REGION Network 66: UNIT 2 STATION 3 COAXIAL CAMERA START NOZZLE ANALISIS METHOD WORKING OR BLOCKED ALARM
   RUNG wire#powerrail
      Contact( "DB16345_U2_STA3_CAM_NOZZLE_ANALISIS_TRIG".Done )
      { S7_Templates := "SrcType := Int" } NE_Contact(in1 := "DB16005_U2_STA3_COAXIAL_CLIENT_INTERFACE".U2_STA3_CAM_Analysis."Analyze nozzle".Outputs.Result, in2 := 0)
      wire#w1
      Contact( "DB7257_UNIT_2_STA_3_COAXIAL_ENABLE_DISABLE".ENABLED )
      wire#w2
      Coil( "DB16000_OPC_UA_TRIGGER_ALARM".CLIENT.U2_STA3_COAXIAL.ALARMS.CAM_START_NOZZLE_ANALISIS_METHOD_WORKING_BLOCKED_A )
   END_RUNG
   RUNG wire#powerrail
      Contact( "DB16000_OPC_UA_TRIGGER_ALARM".CLIENT.U2_STA3_COAXIAL.ALARMS.CAM_START_NOZZLE_ANALISIS_METHOD_WORKING_BLOCKED_A )
      I_Contact( "DB2120_MPP_ITC_IPC".RESET_FAULTS )
   END_RUNG wire#w1
   RUNG wire#w2
      Coil( "DB426_ALARMS_WARNINGS".ALARMS.UNIT_02.STATION_3_COAXIAL."720913" )
   END_RUNG
   // the same network as SCL:
   "DB16000_OPC_UA_TRIGGER_ALARM".CLIENT.U2_STA3_COAXIAL.ALARMS.CAM_START_NOZZLE_ANALISIS_METHOD_WORKING_BLOCKED_A := (("DB16345_U2_STA3_CAM_NOZZLE_ANALISIS_TRIG".Done AND ("DB16005_U2_STA3_COAXIAL_CLIENT_INTERFACE".U2_STA3_CAM_Analysis."Analyze nozzle".Outputs.Result <> 0)) OR ("DB16000_OPC_UA_TRIGGER_ALARM".CLIENT.U2_STA3_COAXIAL.ALARMS.CAM_START_NOZZLE_ANALISIS_METHOD_WORKING_BLOCKED_A AND NOT "DB2120_MPP_ITC_IPC".RESET_FAULTS)) AND "DB7257_UNIT_2_STA_3_COAXIAL_ENABLE_DISABLE".ENABLED;
   "DB426_ALARMS_WARNINGS".ALARMS.UNIT_02.STATION_3_COAXIAL."720913" := "DB16000_OPC_UA_TRIGGER_ALARM".CLIENT.U2_STA3_COAXIAL.ALARMS.CAM_START_NOZZLE_ANALISIS_METHOD_WORKING_BLOCKED_A;
END_REGION

REGION Network 67: UNIT 2 STATION 3 COAXIAL CAMERA START JET ANALISIS METHOD CONNECTION ALARM
   RUNG wire#powerrail
      Contact( "DB16346_U2_STA3_CAM_JET_ANALISIS_TRIG".Error )
      wire#w1
      Contact( "DB7257_UNIT_2_STA_3_COAXIAL_ENABLE_DISABLE".ENABLED )
      wire#w2
      Coil( "DB16000_OPC_UA_TRIGGER_ALARM".CLIENT.U2_STA3_COAXIAL.ALARMS.CAM_START_JET_ANALISIS_CONNECTION_A )
   END_RUNG
   RUNG wire#powerrail
      Contact( "DB16000_OPC_UA_TRIGGER_ALARM".CLIENT.U2_STA3_COAXIAL.ALARMS.CAM_START_JET_ANALISIS_CONNECTION_A )
      I_Contact( "DB2120_MPP_ITC_IPC".RESET_FAULTS )
   END_RUNG wire#w1
   RUNG wire#w2
      Coil( "DB426_ALARMS_WARNINGS".ALARMS.UNIT_02.STATION_3_COAXIAL."720920" )
   END_RUNG
   // the same network as SCL:
   "DB16000_OPC_UA_TRIGGER_ALARM".CLIENT.U2_STA3_COAXIAL.ALARMS.CAM_START_JET_ANALISIS_CONNECTION_A := ("DB16346_U2_STA3_CAM_JET_ANALISIS_TRIG".Error OR ("DB16000_OPC_UA_TRIGGER_ALARM".CLIENT.U2_STA3_COAXIAL.ALARMS.CAM_START_JET_ANALISIS_CONNECTION_A AND NOT "DB2120_MPP_ITC_IPC".RESET_FAULTS)) AND "DB7257_UNIT_2_STA_3_COAXIAL_ENABLE_DISABLE".ENABLED;
   "DB426_ALARMS_WARNINGS".ALARMS.UNIT_02.STATION_3_COAXIAL."720920" := "DB16000_OPC_UA_TRIGGER_ALARM".CLIENT.U2_STA3_COAXIAL.ALARMS.CAM_START_JET_ANALISIS_CONNECTION_A;
END_REGION

REGION Network 68: UNIT 2 STATION 3 COAXIAL CAMERA START JET ANALISIS METHOD WORKING OR BLOCKED ALARM
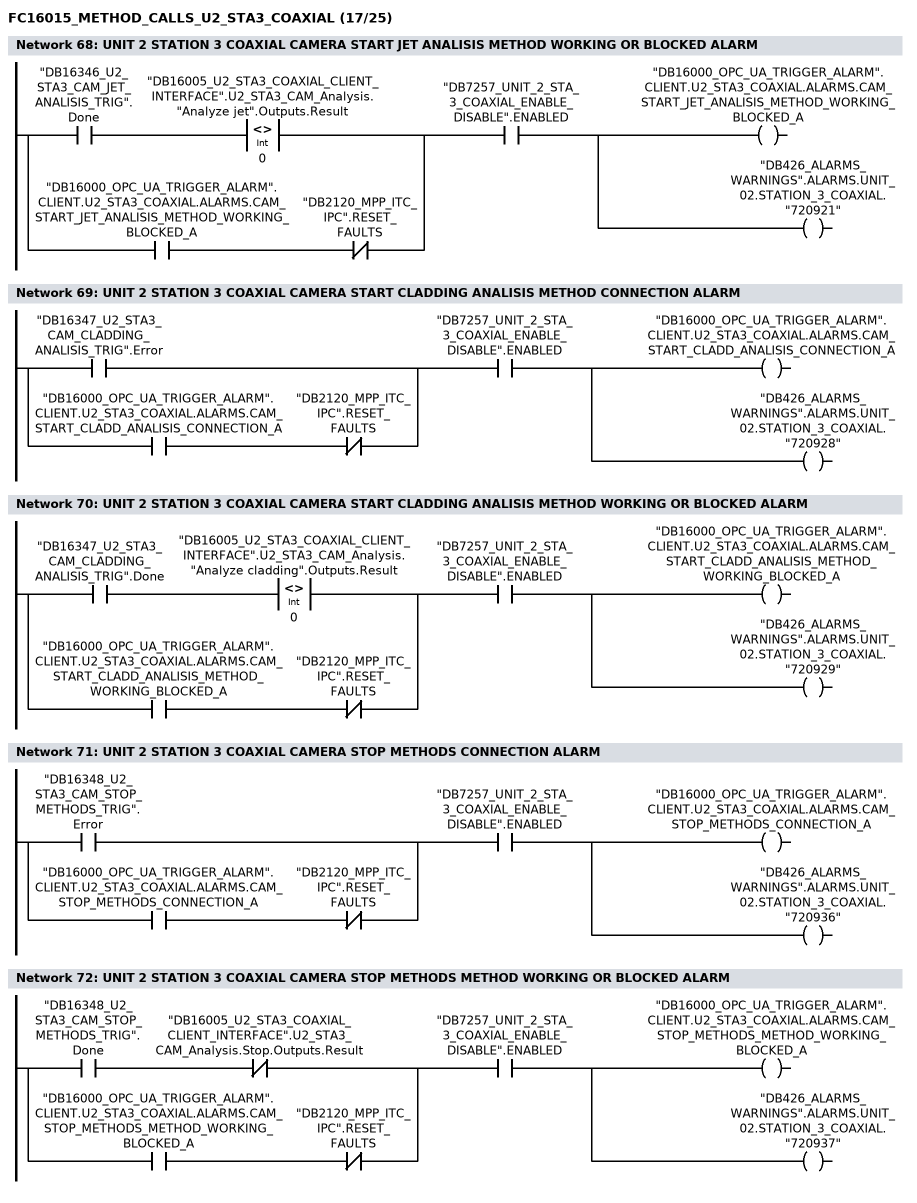
   RUNG wire#powerrail
      Contact( "DB16346_U2_STA3_CAM_JET_ANALISIS_TRIG".Done )
      { S7_Templates := "SrcType := Int" } NE_Contact(in1 := "DB16005_U2_STA3_COAXIAL_CLIENT_INTERFACE".U2_STA3_CAM_Analysis."Analyze jet".Outputs.Result, in2 := 0)
      wire#w1
      Contact( "DB7257_UNIT_2_STA_3_COAXIAL_ENABLE_DISABLE".ENABLED )
      wire#w2
      Coil( "DB16000_OPC_UA_TRIGGER_ALARM".CLIENT.U2_STA3_COAXIAL.ALARMS.CAM_START_JET_ANALISIS_METHOD_WORKING_BLOCKED_A )
   END_RUNG
   RUNG wire#powerrail
      Contact( "DB16000_OPC_UA_TRIGGER_ALARM".CLIENT.U2_STA3_COAXIAL.ALARMS.CAM_START_JET_ANALISIS_METHOD_WORKING_BLOCKED_A )
      I_Contact( "DB2120_MPP_ITC_IPC".RESET_FAULTS )
   END_RUNG wire#w1
   RUNG wire#w2
      Coil( "DB426_ALARMS_WARNINGS".ALARMS.UNIT_02.STATION_3_COAXIAL."720921" )
   END_RUNG
   // the same network as SCL:
   "DB16000_OPC_UA_TRIGGER_ALARM".CLIENT.U2_STA3_COAXIAL.ALARMS.CAM_START_JET_ANALISIS_METHOD_WORKING_BLOCKED_A := (("DB16346_U2_STA3_CAM_JET_ANALISIS_TRIG".Done AND ("DB16005_U2_STA3_COAXIAL_CLIENT_INTERFACE".U2_STA3_CAM_Analysis."Analyze jet".Outputs.Result <> 0)) OR ("DB16000_OPC_UA_TRIGGER_ALARM".CLIENT.U2_STA3_COAXIAL.ALARMS.CAM_START_JET_ANALISIS_METHOD_WORKING_BLOCKED_A AND NOT "DB2120_MPP_ITC_IPC".RESET_FAULTS)) AND "DB7257_UNIT_2_STA_3_COAXIAL_ENABLE_DISABLE".ENABLED;
   "DB426_ALARMS_WARNINGS".ALARMS.UNIT_02.STATION_3_COAXIAL."720921" := "DB16000_OPC_UA_TRIGGER_ALARM".CLIENT.U2_STA3_COAXIAL.ALARMS.CAM_START_JET_ANALISIS_METHOD_WORKING_BLOCKED_A;
END_REGION

REGION Network 69: UNIT 2 STATION 3 COAXIAL CAMERA START CLADDING ANALISIS METHOD CONNECTION ALARM
   RUNG wire#powerrail
      Contact( "DB16347_U2_STA3_CAM_CLADDING_ANALISIS_TRIG".Error )
      wire#w1
      Contact( "DB7257_UNIT_2_STA_3_COAXIAL_ENABLE_DISABLE".ENABLED )
      wire#w2
      Coil( "DB16000_OPC_UA_TRIGGER_ALARM".CLIENT.U2_STA3_COAXIAL.ALARMS.CAM_START_CLADD_ANALISIS_CONNECTION_A )
   END_RUNG
   RUNG wire#powerrail
      Contact( "DB16000_OPC_UA_TRIGGER_ALARM".CLIENT.U2_STA3_COAXIAL.ALARMS.CAM_START_CLADD_ANALISIS_CONNECTION_A )
      I_Contact( "DB2120_MPP_ITC_IPC".RESET_FAULTS )
   END_RUNG wire#w1
   RUNG wire#w2
      Coil( "DB426_ALARMS_WARNINGS".ALARMS.UNIT_02.STATION_3_COAXIAL."720928" )
   END_RUNG
   // the same network as SCL:
   "DB16000_OPC_UA_TRIGGER_ALARM".CLIENT.U2_STA3_COAXIAL.ALARMS.CAM_START_CLADD_ANALISIS_CONNECTION_A := ("DB16347_U2_STA3_CAM_CLADDING_ANALISIS_TRIG".Error OR ("DB16000_OPC_UA_TRIGGER_ALARM".CLIENT.U2_STA3_COAXIAL.ALARMS.CAM_START_CLADD_ANALISIS_CONNECTION_A AND NOT "DB2120_MPP_ITC_IPC".RESET_FAULTS)) AND "DB7257_UNIT_2_STA_3_COAXIAL_ENABLE_DISABLE".ENABLED;
   "DB426_ALARMS_WARNINGS".ALARMS.UNIT_02.STATION_3_COAXIAL."720928" := "DB16000_OPC_UA_TRIGGER_ALARM".CLIENT.U2_STA3_COAXIAL.ALARMS.CAM_START_CLADD_ANALISIS_CONNECTION_A;
END_REGION

REGION Network 70: UNIT 2 STATION 3 COAXIAL CAMERA START CLADDING ANALISIS METHOD WORKING OR BLOCKED ALARM
   RUNG wire#powerrail
      Contact( "DB16347_U2_STA3_CAM_CLADDING_ANALISIS_TRIG".Done )
      { S7_Templates := "SrcType := Int" } NE_Contact(in1 := "DB16005_U2_STA3_COAXIAL_CLIENT_INTERFACE".U2_STA3_CAM_Analysis."Analyze cladding".Outputs.Result, in2 := 0)
      wire#w1
      Contact( "DB7257_UNIT_2_STA_3_COAXIAL_ENABLE_DISABLE".ENABLED )
      wire#w2
      Coil( "DB16000_OPC_UA_TRIGGER_ALARM".CLIENT.U2_STA3_COAXIAL.ALARMS.CAM_START_CLADD_ANALISIS_METHOD_WORKING_BLOCKED_A )
   END_RUNG
   RUNG wire#powerrail
      Contact( "DB16000_OPC_UA_TRIGGER_ALARM".CLIENT.U2_STA3_COAXIAL.ALARMS.CAM_START_CLADD_ANALISIS_METHOD_WORKING_BLOCKED_A )
      I_Contact( "DB2120_MPP_ITC_IPC".RESET_FAULTS )
   END_RUNG wire#w1
   RUNG wire#w2
      Coil( "DB426_ALARMS_WARNINGS".ALARMS.UNIT_02.STATION_3_COAXIAL."720929" )
   END_RUNG
   // the same network as SCL:
   "DB16000_OPC_UA_TRIGGER_ALARM".CLIENT.U2_STA3_COAXIAL.ALARMS.CAM_START_CLADD_ANALISIS_METHOD_WORKING_BLOCKED_A := (("DB16347_U2_STA3_CAM_CLADDING_ANALISIS_TRIG".Done AND ("DB16005_U2_STA3_COAXIAL_CLIENT_INTERFACE".U2_STA3_CAM_Analysis."Analyze cladding".Outputs.Result <> 0)) OR ("DB16000_OPC_UA_TRIGGER_ALARM".CLIENT.U2_STA3_COAXIAL.ALARMS.CAM_START_CLADD_ANALISIS_METHOD_WORKING_BLOCKED_A AND NOT "DB2120_MPP_ITC_IPC".RESET_FAULTS)) AND "DB7257_UNIT_2_STA_3_COAXIAL_ENABLE_DISABLE".ENABLED;
   "DB426_ALARMS_WARNINGS".ALARMS.UNIT_02.STATION_3_COAXIAL."720929" := "DB16000_OPC_UA_TRIGGER_ALARM".CLIENT.U2_STA3_COAXIAL.ALARMS.CAM_START_CLADD_ANALISIS_METHOD_WORKING_BLOCKED_A;
END_REGION

REGION Network 71: UNIT 2 STATION 3 COAXIAL CAMERA STOP METHODS CONNECTION ALARM
   RUNG wire#powerrail
      Contact( "DB16348_U2_STA3_CAM_STOP_METHODS_TRIG".Error )
      wire#w1
      Contact( "DB7257_UNIT_2_STA_3_COAXIAL_ENABLE_DISABLE".ENABLED )
      wire#w2
      Coil( "DB16000_OPC_UA_TRIGGER_ALARM".CLIENT.U2_STA3_COAXIAL.ALARMS.CAM_STOP_METHODS_CONNECTION_A )
   END_RUNG
   RUNG wire#powerrail
      Contact( "DB16000_OPC_UA_TRIGGER_ALARM".CLIENT.U2_STA3_COAXIAL.ALARMS.CAM_STOP_METHODS_CONNECTION_A )
      I_Contact( "DB2120_MPP_ITC_IPC".RESET_FAULTS )
   END_RUNG wire#w1
   RUNG wire#w2
      Coil( "DB426_ALARMS_WARNINGS".ALARMS.UNIT_02.STATION_3_COAXIAL."720936" )
   END_RUNG
   // the same network as SCL:
   "DB16000_OPC_UA_TRIGGER_ALARM".CLIENT.U2_STA3_COAXIAL.ALARMS.CAM_STOP_METHODS_CONNECTION_A := ("DB16348_U2_STA3_CAM_STOP_METHODS_TRIG".Error OR ("DB16000_OPC_UA_TRIGGER_ALARM".CLIENT.U2_STA3_COAXIAL.ALARMS.CAM_STOP_METHODS_CONNECTION_A AND NOT "DB2120_MPP_ITC_IPC".RESET_FAULTS)) AND "DB7257_UNIT_2_STA_3_COAXIAL_ENABLE_DISABLE".ENABLED;
   "DB426_ALARMS_WARNINGS".ALARMS.UNIT_02.STATION_3_COAXIAL."720936" := "DB16000_OPC_UA_TRIGGER_ALARM".CLIENT.U2_STA3_COAXIAL.ALARMS.CAM_STOP_METHODS_CONNECTION_A;
END_REGION

REGION Network 72: UNIT 2 STATION 3 COAXIAL CAMERA STOP METHODS METHOD WORKING OR BLOCKED ALARM
   RUNG wire#powerrail
      Contact( "DB16348_U2_STA3_CAM_STOP_METHODS_TRIG".Done )
      I_Contact( "DB16005_U2_STA3_COAXIAL_CLIENT_INTERFACE".U2_STA3_CAM_Analysis.Stop.Outputs.Result )
      wire#w1
      Contact( "DB7257_UNIT_2_STA_3_COAXIAL_ENABLE_DISABLE".ENABLED )
      wire#w2
      Coil( "DB16000_OPC_UA_TRIGGER_ALARM".CLIENT.U2_STA3_COAXIAL.ALARMS.CAM_STOP_METHODS_METHOD_WORKING_BLOCKED_A )
   END_RUNG
   RUNG wire#powerrail
      Contact( "DB16000_OPC_UA_TRIGGER_ALARM".CLIENT.U2_STA3_COAXIAL.ALARMS.CAM_STOP_METHODS_METHOD_WORKING_BLOCKED_A )
      I_Contact( "DB2120_MPP_ITC_IPC".RESET_FAULTS )
   END_RUNG wire#w1
   RUNG wire#w2
      Coil( "DB426_ALARMS_WARNINGS".ALARMS.UNIT_02.STATION_3_COAXIAL."720937" )
   END_RUNG
   // the same network as SCL:
   "DB16000_OPC_UA_TRIGGER_ALARM".CLIENT.U2_STA3_COAXIAL.ALARMS.CAM_STOP_METHODS_METHOD_WORKING_BLOCKED_A := (("DB16348_U2_STA3_CAM_STOP_METHODS_TRIG".Done AND NOT "DB16005_U2_STA3_COAXIAL_CLIENT_INTERFACE".U2_STA3_CAM_Analysis.Stop.Outputs.Result) OR ("DB16000_OPC_UA_TRIGGER_ALARM".CLIENT.U2_STA3_COAXIAL.ALARMS.CAM_STOP_METHODS_METHOD_WORKING_BLOCKED_A AND NOT "DB2120_MPP_ITC_IPC".RESET_FAULTS)) AND "DB7257_UNIT_2_STA_3_COAXIAL_ENABLE_DISABLE".ENABLED;
   "DB426_ALARMS_WARNINGS".ALARMS.UNIT_02.STATION_3_COAXIAL."720937" := "DB16000_OPC_UA_TRIGGER_ALARM".CLIENT.U2_STA3_COAXIAL.ALARMS.CAM_STOP_METHODS_METHOD_WORKING_BLOCKED_A;
END_REGION

REGION Network 73: UNIT 2 STATION 3 COAXIAL CAMERA RESET PC METHOD CONNECTION ALARM
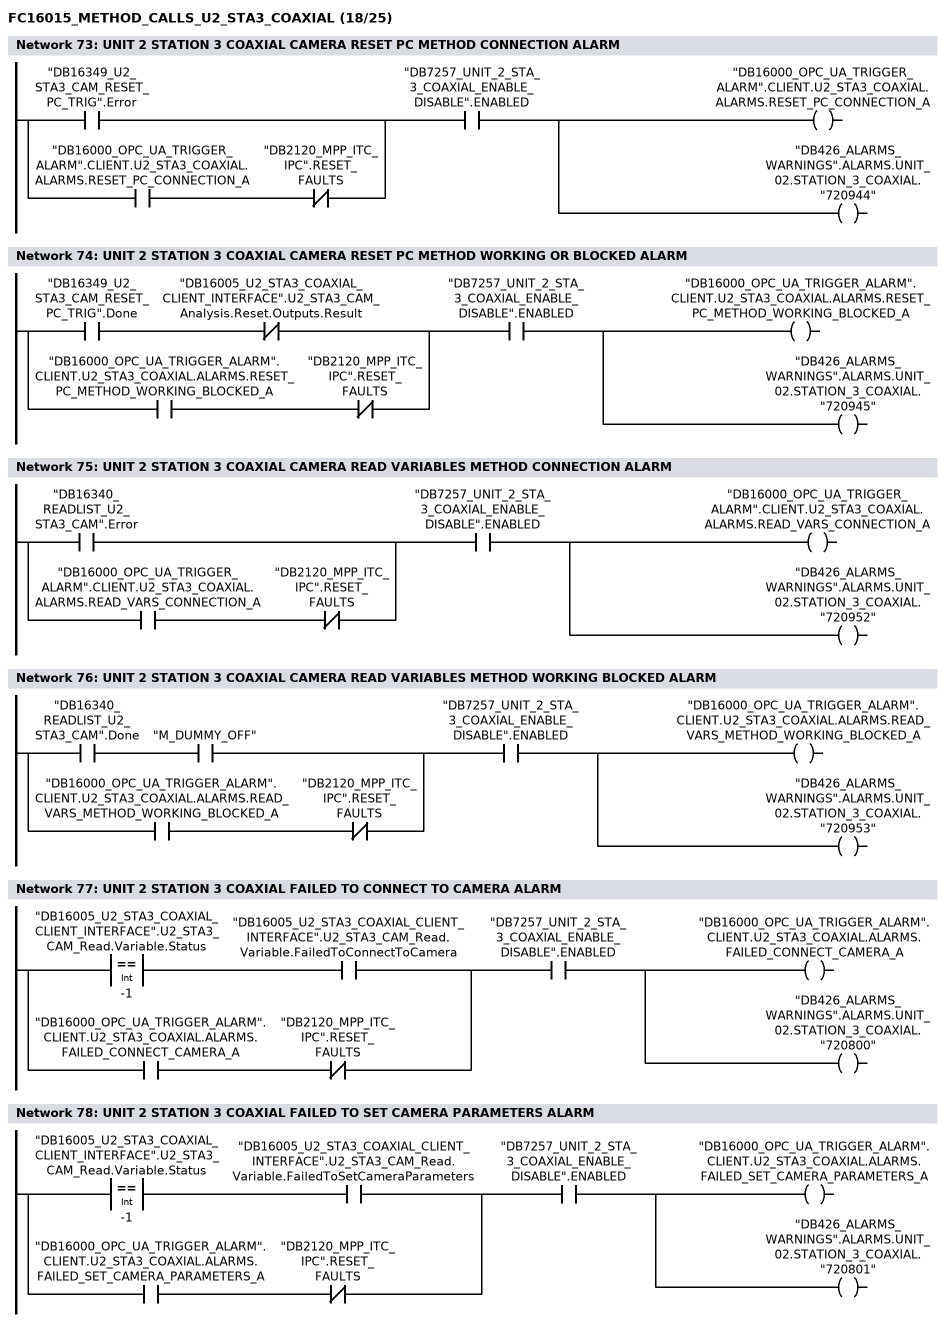
   RUNG wire#powerrail
      Contact( "DB16349_U2_STA3_CAM_RESET_PC_TRIG".Error )
      wire#w1
      Contact( "DB7257_UNIT_2_STA_3_COAXIAL_ENABLE_DISABLE".ENABLED )
      wire#w2
      Coil( "DB16000_OPC_UA_TRIGGER_ALARM".CLIENT.U2_STA3_COAXIAL.ALARMS.RESET_PC_CONNECTION_A )
   END_RUNG
   RUNG wire#powerrail
      Contact( "DB16000_OPC_UA_TRIGGER_ALARM".CLIENT.U2_STA3_COAXIAL.ALARMS.RESET_PC_CONNECTION_A )
      I_Contact( "DB2120_MPP_ITC_IPC".RESET_FAULTS )
   END_RUNG wire#w1
   RUNG wire#w2
      Coil( "DB426_ALARMS_WARNINGS".ALARMS.UNIT_02.STATION_3_COAXIAL."720944" )
   END_RUNG
   // the same network as SCL:
   "DB16000_OPC_UA_TRIGGER_ALARM".CLIENT.U2_STA3_COAXIAL.ALARMS.RESET_PC_CONNECTION_A := ("DB16349_U2_STA3_CAM_RESET_PC_TRIG".Error OR ("DB16000_OPC_UA_TRIGGER_ALARM".CLIENT.U2_STA3_COAXIAL.ALARMS.RESET_PC_CONNECTION_A AND NOT "DB2120_MPP_ITC_IPC".RESET_FAULTS)) AND "DB7257_UNIT_2_STA_3_COAXIAL_ENABLE_DISABLE".ENABLED;
   "DB426_ALARMS_WARNINGS".ALARMS.UNIT_02.STATION_3_COAXIAL."720944" := "DB16000_OPC_UA_TRIGGER_ALARM".CLIENT.U2_STA3_COAXIAL.ALARMS.RESET_PC_CONNECTION_A;
END_REGION

REGION Network 74: UNIT 2 STATION 3 COAXIAL CAMERA RESET PC METHOD WORKING OR BLOCKED ALARM
   RUNG wire#powerrail
      Contact( "DB16349_U2_STA3_CAM_RESET_PC_TRIG".Done )
      I_Contact( "DB16005_U2_STA3_COAXIAL_CLIENT_INTERFACE".U2_STA3_CAM_Analysis.Reset.Outputs.Result )
      wire#w1
      Contact( "DB7257_UNIT_2_STA_3_COAXIAL_ENABLE_DISABLE".ENABLED )
      wire#w2
      Coil( "DB16000_OPC_UA_TRIGGER_ALARM".CLIENT.U2_STA3_COAXIAL.ALARMS.RESET_PC_METHOD_WORKING_BLOCKED_A )
   END_RUNG
   RUNG wire#powerrail
      Contact( "DB16000_OPC_UA_TRIGGER_ALARM".CLIENT.U2_STA3_COAXIAL.ALARMS.RESET_PC_METHOD_WORKING_BLOCKED_A )
      I_Contact( "DB2120_MPP_ITC_IPC".RESET_FAULTS )
   END_RUNG wire#w1
   RUNG wire#w2
      Coil( "DB426_ALARMS_WARNINGS".ALARMS.UNIT_02.STATION_3_COAXIAL."720945" )
   END_RUNG
   // the same network as SCL:
   "DB16000_OPC_UA_TRIGGER_ALARM".CLIENT.U2_STA3_COAXIAL.ALARMS.RESET_PC_METHOD_WORKING_BLOCKED_A := (("DB16349_U2_STA3_CAM_RESET_PC_TRIG".Done AND NOT "DB16005_U2_STA3_COAXIAL_CLIENT_INTERFACE".U2_STA3_CAM_Analysis.Reset.Outputs.Result) OR ("DB16000_OPC_UA_TRIGGER_ALARM".CLIENT.U2_STA3_COAXIAL.ALARMS.RESET_PC_METHOD_WORKING_BLOCKED_A AND NOT "DB2120_MPP_ITC_IPC".RESET_FAULTS)) AND "DB7257_UNIT_2_STA_3_COAXIAL_ENABLE_DISABLE".ENABLED;
   "DB426_ALARMS_WARNINGS".ALARMS.UNIT_02.STATION_3_COAXIAL."720945" := "DB16000_OPC_UA_TRIGGER_ALARM".CLIENT.U2_STA3_COAXIAL.ALARMS.RESET_PC_METHOD_WORKING_BLOCKED_A;
END_REGION

REGION Network 75: UNIT 2 STATION 3 COAXIAL CAMERA READ VARIABLES METHOD CONNECTION ALARM
   RUNG wire#powerrail
      Contact( "DB16340_READLIST_U2_STA3_CAM".Error )
      wire#w1
      Contact( "DB7257_UNIT_2_STA_3_COAXIAL_ENABLE_DISABLE".ENABLED )
      wire#w2
      Coil( "DB16000_OPC_UA_TRIGGER_ALARM".CLIENT.U2_STA3_COAXIAL.ALARMS.READ_VARS_CONNECTION_A )
   END_RUNG
   RUNG wire#powerrail
      Contact( "DB16000_OPC_UA_TRIGGER_ALARM".CLIENT.U2_STA3_COAXIAL.ALARMS.READ_VARS_CONNECTION_A )
      I_Contact( "DB2120_MPP_ITC_IPC".RESET_FAULTS )
   END_RUNG wire#w1
   RUNG wire#w2
      Coil( "DB426_ALARMS_WARNINGS".ALARMS.UNIT_02.STATION_3_COAXIAL."720952" )
   END_RUNG
   // the same network as SCL:
   "DB16000_OPC_UA_TRIGGER_ALARM".CLIENT.U2_STA3_COAXIAL.ALARMS.READ_VARS_CONNECTION_A := ("DB16340_READLIST_U2_STA3_CAM".Error OR ("DB16000_OPC_UA_TRIGGER_ALARM".CLIENT.U2_STA3_COAXIAL.ALARMS.READ_VARS_CONNECTION_A AND NOT "DB2120_MPP_ITC_IPC".RESET_FAULTS)) AND "DB7257_UNIT_2_STA_3_COAXIAL_ENABLE_DISABLE".ENABLED;
   "DB426_ALARMS_WARNINGS".ALARMS.UNIT_02.STATION_3_COAXIAL."720952" := "DB16000_OPC_UA_TRIGGER_ALARM".CLIENT.U2_STA3_COAXIAL.ALARMS.READ_VARS_CONNECTION_A;
END_REGION

REGION Network 76: UNIT 2 STATION 3 COAXIAL CAMERA READ VARIABLES METHOD WORKING BLOCKED ALARM
   RUNG wire#powerrail
      Contact( "DB16340_READLIST_U2_STA3_CAM".Done )
      Contact( "M_DUMMY_OFF" )
      wire#w1
      Contact( "DB7257_UNIT_2_STA_3_COAXIAL_ENABLE_DISABLE".ENABLED )
      wire#w2
      Coil( "DB16000_OPC_UA_TRIGGER_ALARM".CLIENT.U2_STA3_COAXIAL.ALARMS.READ_VARS_METHOD_WORKING_BLOCKED_A )
   END_RUNG
   RUNG wire#powerrail
      Contact( "DB16000_OPC_UA_TRIGGER_ALARM".CLIENT.U2_STA3_COAXIAL.ALARMS.READ_VARS_METHOD_WORKING_BLOCKED_A )
      I_Contact( "DB2120_MPP_ITC_IPC".RESET_FAULTS )
   END_RUNG wire#w1
   RUNG wire#w2
      Coil( "DB426_ALARMS_WARNINGS".ALARMS.UNIT_02.STATION_3_COAXIAL."720953" )
   END_RUNG
   // the same network as SCL:
   "DB16000_OPC_UA_TRIGGER_ALARM".CLIENT.U2_STA3_COAXIAL.ALARMS.READ_VARS_METHOD_WORKING_BLOCKED_A := (("DB16340_READLIST_U2_STA3_CAM".Done AND "M_DUMMY_OFF") OR ("DB16000_OPC_UA_TRIGGER_ALARM".CLIENT.U2_STA3_COAXIAL.ALARMS.READ_VARS_METHOD_WORKING_BLOCKED_A AND NOT "DB2120_MPP_ITC_IPC".RESET_FAULTS)) AND "DB7257_UNIT_2_STA_3_COAXIAL_ENABLE_DISABLE".ENABLED;
   "DB426_ALARMS_WARNINGS".ALARMS.UNIT_02.STATION_3_COAXIAL."720953" := "DB16000_OPC_UA_TRIGGER_ALARM".CLIENT.U2_STA3_COAXIAL.ALARMS.READ_VARS_METHOD_WORKING_BLOCKED_A;
END_REGION

REGION Network 77: UNIT 2 STATION 3 COAXIAL FAILED TO CONNECT TO CAMERA ALARM
   RUNG wire#powerrail
      { S7_Templates := "SrcType := Int" } EQ_Contact(in1 := "DB16005_U2_STA3_COAXIAL_CLIENT_INTERFACE".U2_STA3_CAM_Read.Variable.Status, in2 := -1)
      Contact( "DB16005_U2_STA3_COAXIAL_CLIENT_INTERFACE".U2_STA3_CAM_Read.Variable.FailedToConnectToCamera )
      wire#w1
      Contact( "DB7257_UNIT_2_STA_3_COAXIAL_ENABLE_DISABLE".ENABLED )
      wire#w2
      Coil( "DB16000_OPC_UA_TRIGGER_ALARM".CLIENT.U2_STA3_COAXIAL.ALARMS.FAILED_CONNECT_CAMERA_A )
   END_RUNG
   RUNG wire#powerrail
      Contact( "DB16000_OPC_UA_TRIGGER_ALARM".CLIENT.U2_STA3_COAXIAL.ALARMS.FAILED_CONNECT_CAMERA_A )
      I_Contact( "DB2120_MPP_ITC_IPC".RESET_FAULTS )
   END_RUNG wire#w1
   RUNG wire#w2
      Coil( "DB426_ALARMS_WARNINGS".ALARMS.UNIT_02.STATION_3_COAXIAL."720800" )
   END_RUNG
   // the same network as SCL:
   "DB16000_OPC_UA_TRIGGER_ALARM".CLIENT.U2_STA3_COAXIAL.ALARMS.FAILED_CONNECT_CAMERA_A := ((("DB16005_U2_STA3_COAXIAL_CLIENT_INTERFACE".U2_STA3_CAM_Read.Variable.Status = (-1)) AND "DB16005_U2_STA3_COAXIAL_CLIENT_INTERFACE".U2_STA3_CAM_Read.Variable.FailedToConnectToCamera) OR ("DB16000_OPC_UA_TRIGGER_ALARM".CLIENT.U2_STA3_COAXIAL.ALARMS.FAILED_CONNECT_CAMERA_A AND NOT "DB2120_MPP_ITC_IPC".RESET_FAULTS)) AND "DB7257_UNIT_2_STA_3_COAXIAL_ENABLE_DISABLE".ENABLED;
   "DB426_ALARMS_WARNINGS".ALARMS.UNIT_02.STATION_3_COAXIAL."720800" := "DB16000_OPC_UA_TRIGGER_ALARM".CLIENT.U2_STA3_COAXIAL.ALARMS.FAILED_CONNECT_CAMERA_A;
END_REGION

REGION Network 78: UNIT 2 STATION 3 COAXIAL FAILED TO SET CAMERA PARAMETERS ALARM
   RUNG wire#powerrail
      { S7_Templates := "SrcType := Int" } EQ_Contact(in1 := "DB16005_U2_STA3_COAXIAL_CLIENT_INTERFACE".U2_STA3_CAM_Read.Variable.Status, in2 := -1)
      Contact( "DB16005_U2_STA3_COAXIAL_CLIENT_INTERFACE".U2_STA3_CAM_Read.Variable.FailedToSetCameraParameters )
      wire#w1
      Contact( "DB7257_UNIT_2_STA_3_COAXIAL_ENABLE_DISABLE".ENABLED )
      wire#w2
      Coil( "DB16000_OPC_UA_TRIGGER_ALARM".CLIENT.U2_STA3_COAXIAL.ALARMS.FAILED_SET_CAMERA_PARAMETERS_A )
   END_RUNG
   RUNG wire#powerrail
      Contact( "DB16000_OPC_UA_TRIGGER_ALARM".CLIENT.U2_STA3_COAXIAL.ALARMS.FAILED_SET_CAMERA_PARAMETERS_A )
      I_Contact( "DB2120_MPP_ITC_IPC".RESET_FAULTS )
   END_RUNG wire#w1
   RUNG wire#w2
      Coil( "DB426_ALARMS_WARNINGS".ALARMS.UNIT_02.STATION_3_COAXIAL."720801" )
   END_RUNG
   // the same network as SCL:
   "DB16000_OPC_UA_TRIGGER_ALARM".CLIENT.U2_STA3_COAXIAL.ALARMS.FAILED_SET_CAMERA_PARAMETERS_A := ((("DB16005_U2_STA3_COAXIAL_CLIENT_INTERFACE".U2_STA3_CAM_Read.Variable.Status = (-1)) AND "DB16005_U2_STA3_COAXIAL_CLIENT_INTERFACE".U2_STA3_CAM_Read.Variable.FailedToSetCameraParameters) OR ("DB16000_OPC_UA_TRIGGER_ALARM".CLIENT.U2_STA3_COAXIAL.ALARMS.FAILED_SET_CAMERA_PARAMETERS_A AND NOT "DB2120_MPP_ITC_IPC".RESET_FAULTS)) AND "DB7257_UNIT_2_STA_3_COAXIAL_ENABLE_DISABLE".ENABLED;
   "DB426_ALARMS_WARNINGS".ALARMS.UNIT_02.STATION_3_COAXIAL."720801" := "DB16000_OPC_UA_TRIGGER_ALARM".CLIENT.U2_STA3_COAXIAL.ALARMS.FAILED_SET_CAMERA_PARAMETERS_A;
END_REGION

REGION Network 79: UNIT 2 STATION 3 COAXIAL NEW LASER CALIBRATION REQUIERED ALARM
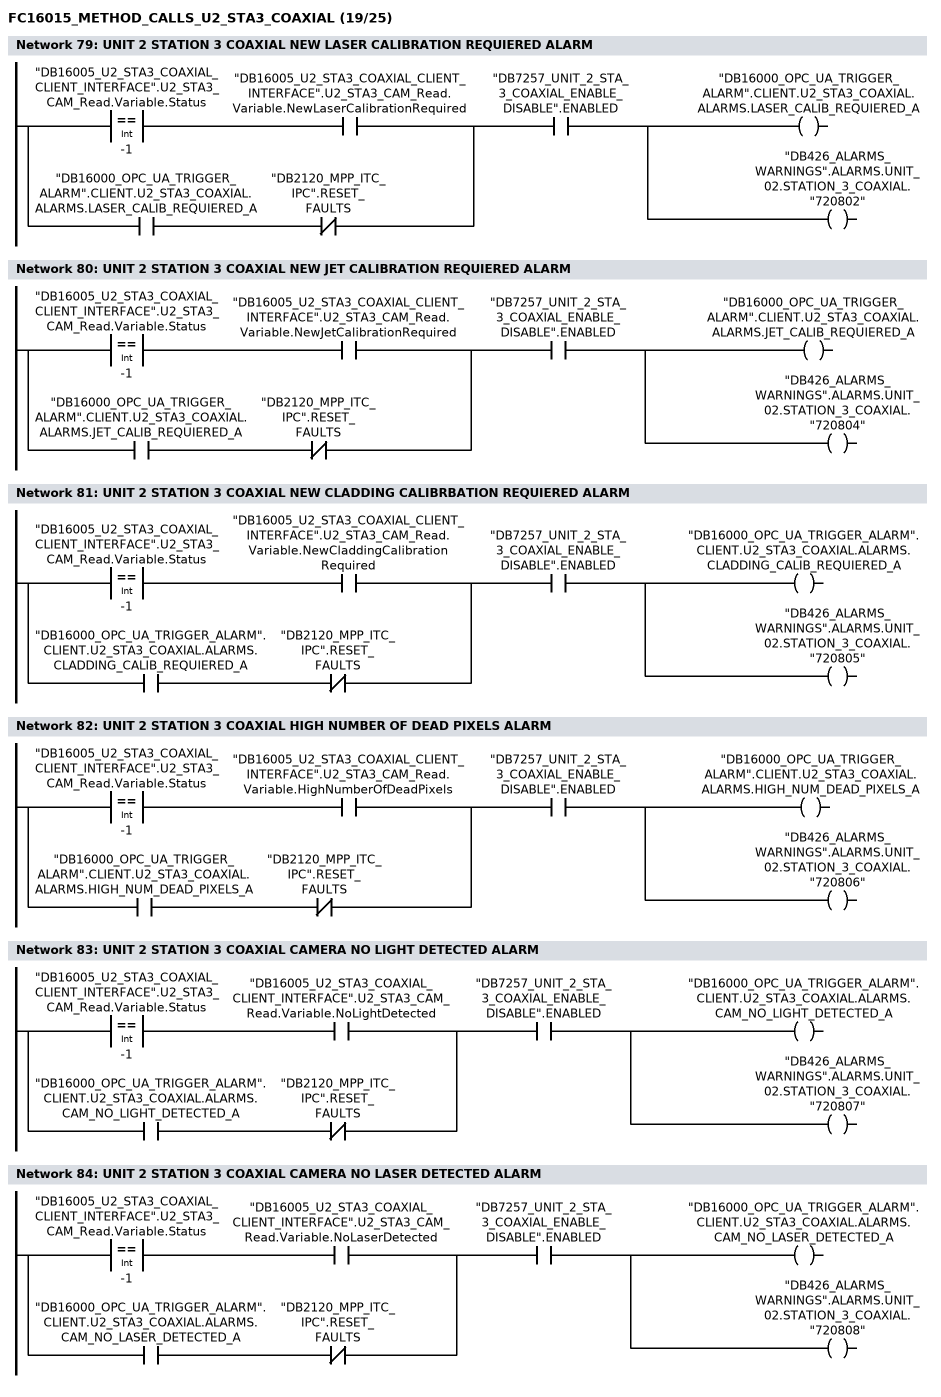
   RUNG wire#powerrail
      { S7_Templates := "SrcType := Int" } EQ_Contact(in1 := "DB16005_U2_STA3_COAXIAL_CLIENT_INTERFACE".U2_STA3_CAM_Read.Variable.Status, in2 := -1)
      Contact( "DB16005_U2_STA3_COAXIAL_CLIENT_INTERFACE".U2_STA3_CAM_Read.Variable.NewLaserCalibrationRequired )
      wire#w1
      Contact( "DB7257_UNIT_2_STA_3_COAXIAL_ENABLE_DISABLE".ENABLED )
      wire#w2
      Coil( "DB16000_OPC_UA_TRIGGER_ALARM".CLIENT.U2_STA3_COAXIAL.ALARMS.LASER_CALIB_REQUIERED_A )
   END_RUNG
   RUNG wire#powerrail
      Contact( "DB16000_OPC_UA_TRIGGER_ALARM".CLIENT.U2_STA3_COAXIAL.ALARMS.LASER_CALIB_REQUIERED_A )
      I_Contact( "DB2120_MPP_ITC_IPC".RESET_FAULTS )
   END_RUNG wire#w1
   RUNG wire#w2
      Coil( "DB426_ALARMS_WARNINGS".ALARMS.UNIT_02.STATION_3_COAXIAL."720802" )
   END_RUNG
   // the same network as SCL:
   "DB16000_OPC_UA_TRIGGER_ALARM".CLIENT.U2_STA3_COAXIAL.ALARMS.LASER_CALIB_REQUIERED_A := ((("DB16005_U2_STA3_COAXIAL_CLIENT_INTERFACE".U2_STA3_CAM_Read.Variable.Status = (-1)) AND "DB16005_U2_STA3_COAXIAL_CLIENT_INTERFACE".U2_STA3_CAM_Read.Variable.NewLaserCalibrationRequired) OR ("DB16000_OPC_UA_TRIGGER_ALARM".CLIENT.U2_STA3_COAXIAL.ALARMS.LASER_CALIB_REQUIERED_A AND NOT "DB2120_MPP_ITC_IPC".RESET_FAULTS)) AND "DB7257_UNIT_2_STA_3_COAXIAL_ENABLE_DISABLE".ENABLED;
   "DB426_ALARMS_WARNINGS".ALARMS.UNIT_02.STATION_3_COAXIAL."720802" := "DB16000_OPC_UA_TRIGGER_ALARM".CLIENT.U2_STA3_COAXIAL.ALARMS.LASER_CALIB_REQUIERED_A;
END_REGION

REGION Network 80: UNIT 2 STATION 3 COAXIAL NEW JET CALIBRATION REQUIERED ALARM
   RUNG wire#powerrail
      { S7_Templates := "SrcType := Int" } EQ_Contact(in1 := "DB16005_U2_STA3_COAXIAL_CLIENT_INTERFACE".U2_STA3_CAM_Read.Variable.Status, in2 := -1)
      Contact( "DB16005_U2_STA3_COAXIAL_CLIENT_INTERFACE".U2_STA3_CAM_Read.Variable.NewJetCalibrationRequired )
      wire#w1
      Contact( "DB7257_UNIT_2_STA_3_COAXIAL_ENABLE_DISABLE".ENABLED )
      wire#w2
      Coil( "DB16000_OPC_UA_TRIGGER_ALARM".CLIENT.U2_STA3_COAXIAL.ALARMS.JET_CALIB_REQUIERED_A )
   END_RUNG
   RUNG wire#powerrail
      Contact( "DB16000_OPC_UA_TRIGGER_ALARM".CLIENT.U2_STA3_COAXIAL.ALARMS.JET_CALIB_REQUIERED_A )
      I_Contact( "DB2120_MPP_ITC_IPC".RESET_FAULTS )
   END_RUNG wire#w1
   RUNG wire#w2
      Coil( "DB426_ALARMS_WARNINGS".ALARMS.UNIT_02.STATION_3_COAXIAL."720804" )
   END_RUNG
   // the same network as SCL:
   "DB16000_OPC_UA_TRIGGER_ALARM".CLIENT.U2_STA3_COAXIAL.ALARMS.JET_CALIB_REQUIERED_A := ((("DB16005_U2_STA3_COAXIAL_CLIENT_INTERFACE".U2_STA3_CAM_Read.Variable.Status = (-1)) AND "DB16005_U2_STA3_COAXIAL_CLIENT_INTERFACE".U2_STA3_CAM_Read.Variable.NewJetCalibrationRequired) OR ("DB16000_OPC_UA_TRIGGER_ALARM".CLIENT.U2_STA3_COAXIAL.ALARMS.JET_CALIB_REQUIERED_A AND NOT "DB2120_MPP_ITC_IPC".RESET_FAULTS)) AND "DB7257_UNIT_2_STA_3_COAXIAL_ENABLE_DISABLE".ENABLED;
   "DB426_ALARMS_WARNINGS".ALARMS.UNIT_02.STATION_3_COAXIAL."720804" := "DB16000_OPC_UA_TRIGGER_ALARM".CLIENT.U2_STA3_COAXIAL.ALARMS.JET_CALIB_REQUIERED_A;
END_REGION

REGION Network 81: UNIT 2 STATION 3 COAXIAL NEW CLADDING CALIBRBATION REQUIERED ALARM
   RUNG wire#powerrail
      { S7_Templates := "SrcType := Int" } EQ_Contact(in1 := "DB16005_U2_STA3_COAXIAL_CLIENT_INTERFACE".U2_STA3_CAM_Read.Variable.Status, in2 := -1)
      Contact( "DB16005_U2_STA3_COAXIAL_CLIENT_INTERFACE".U2_STA3_CAM_Read.Variable.NewCladdingCalibrationRequired )
      wire#w1
      Contact( "DB7257_UNIT_2_STA_3_COAXIAL_ENABLE_DISABLE".ENABLED )
      wire#w2
      Coil( "DB16000_OPC_UA_TRIGGER_ALARM".CLIENT.U2_STA3_COAXIAL.ALARMS.CLADDING_CALIB_REQUIERED_A )
   END_RUNG
   RUNG wire#powerrail
      Contact( "DB16000_OPC_UA_TRIGGER_ALARM".CLIENT.U2_STA3_COAXIAL.ALARMS.CLADDING_CALIB_REQUIERED_A )
      I_Contact( "DB2120_MPP_ITC_IPC".RESET_FAULTS )
   END_RUNG wire#w1
   RUNG wire#w2
      Coil( "DB426_ALARMS_WARNINGS".ALARMS.UNIT_02.STATION_3_COAXIAL."720805" )
   END_RUNG
   // the same network as SCL:
   "DB16000_OPC_UA_TRIGGER_ALARM".CLIENT.U2_STA3_COAXIAL.ALARMS.CLADDING_CALIB_REQUIERED_A := ((("DB16005_U2_STA3_COAXIAL_CLIENT_INTERFACE".U2_STA3_CAM_Read.Variable.Status = (-1)) AND "DB16005_U2_STA3_COAXIAL_CLIENT_INTERFACE".U2_STA3_CAM_Read.Variable.NewCladdingCalibrationRequired) OR ("DB16000_OPC_UA_TRIGGER_ALARM".CLIENT.U2_STA3_COAXIAL.ALARMS.CLADDING_CALIB_REQUIERED_A AND NOT "DB2120_MPP_ITC_IPC".RESET_FAULTS)) AND "DB7257_UNIT_2_STA_3_COAXIAL_ENABLE_DISABLE".ENABLED;
   "DB426_ALARMS_WARNINGS".ALARMS.UNIT_02.STATION_3_COAXIAL."720805" := "DB16000_OPC_UA_TRIGGER_ALARM".CLIENT.U2_STA3_COAXIAL.ALARMS.CLADDING_CALIB_REQUIERED_A;
END_REGION

REGION Network 82: UNIT 2 STATION 3 COAXIAL HIGH NUMBER OF DEAD PIXELS ALARM
   RUNG wire#powerrail
      { S7_Templates := "SrcType := Int" } EQ_Contact(in1 := "DB16005_U2_STA3_COAXIAL_CLIENT_INTERFACE".U2_STA3_CAM_Read.Variable.Status, in2 := -1)
      Contact( "DB16005_U2_STA3_COAXIAL_CLIENT_INTERFACE".U2_STA3_CAM_Read.Variable.HighNumberOfDeadPixels )
      wire#w1
      Contact( "DB7257_UNIT_2_STA_3_COAXIAL_ENABLE_DISABLE".ENABLED )
      wire#w2
      Coil( "DB16000_OPC_UA_TRIGGER_ALARM".CLIENT.U2_STA3_COAXIAL.ALARMS.HIGH_NUM_DEAD_PIXELS_A )
   END_RUNG
   RUNG wire#powerrail
      Contact( "DB16000_OPC_UA_TRIGGER_ALARM".CLIENT.U2_STA3_COAXIAL.ALARMS.HIGH_NUM_DEAD_PIXELS_A )
      I_Contact( "DB2120_MPP_ITC_IPC".RESET_FAULTS )
   END_RUNG wire#w1
   RUNG wire#w2
      Coil( "DB426_ALARMS_WARNINGS".ALARMS.UNIT_02.STATION_3_COAXIAL."720806" )
   END_RUNG
   // the same network as SCL:
   "DB16000_OPC_UA_TRIGGER_ALARM".CLIENT.U2_STA3_COAXIAL.ALARMS.HIGH_NUM_DEAD_PIXELS_A := ((("DB16005_U2_STA3_COAXIAL_CLIENT_INTERFACE".U2_STA3_CAM_Read.Variable.Status = (-1)) AND "DB16005_U2_STA3_COAXIAL_CLIENT_INTERFACE".U2_STA3_CAM_Read.Variable.HighNumberOfDeadPixels) OR ("DB16000_OPC_UA_TRIGGER_ALARM".CLIENT.U2_STA3_COAXIAL.ALARMS.HIGH_NUM_DEAD_PIXELS_A AND NOT "DB2120_MPP_ITC_IPC".RESET_FAULTS)) AND "DB7257_UNIT_2_STA_3_COAXIAL_ENABLE_DISABLE".ENABLED;
   "DB426_ALARMS_WARNINGS".ALARMS.UNIT_02.STATION_3_COAXIAL."720806" := "DB16000_OPC_UA_TRIGGER_ALARM".CLIENT.U2_STA3_COAXIAL.ALARMS.HIGH_NUM_DEAD_PIXELS_A;
END_REGION

REGION Network 83: UNIT 2 STATION 3 COAXIAL CAMERA NO LIGHT DETECTED ALARM
   RUNG wire#powerrail
      { S7_Templates := "SrcType := Int" } EQ_Contact(in1 := "DB16005_U2_STA3_COAXIAL_CLIENT_INTERFACE".U2_STA3_CAM_Read.Variable.Status, in2 := -1)
      Contact( "DB16005_U2_STA3_COAXIAL_CLIENT_INTERFACE".U2_STA3_CAM_Read.Variable.NoLightDetected )
      wire#w1
      Contact( "DB7257_UNIT_2_STA_3_COAXIAL_ENABLE_DISABLE".ENABLED )
      wire#w2
      Coil( "DB16000_OPC_UA_TRIGGER_ALARM".CLIENT.U2_STA3_COAXIAL.ALARMS.CAM_NO_LIGHT_DETECTED_A )
   END_RUNG
   RUNG wire#powerrail
      Contact( "DB16000_OPC_UA_TRIGGER_ALARM".CLIENT.U2_STA3_COAXIAL.ALARMS.CAM_NO_LIGHT_DETECTED_A )
      I_Contact( "DB2120_MPP_ITC_IPC".RESET_FAULTS )
   END_RUNG wire#w1
   RUNG wire#w2
      Coil( "DB426_ALARMS_WARNINGS".ALARMS.UNIT_02.STATION_3_COAXIAL."720807" )
   END_RUNG
   // the same network as SCL:
   "DB16000_OPC_UA_TRIGGER_ALARM".CLIENT.U2_STA3_COAXIAL.ALARMS.CAM_NO_LIGHT_DETECTED_A := ((("DB16005_U2_STA3_COAXIAL_CLIENT_INTERFACE".U2_STA3_CAM_Read.Variable.Status = (-1)) AND "DB16005_U2_STA3_COAXIAL_CLIENT_INTERFACE".U2_STA3_CAM_Read.Variable.NoLightDetected) OR ("DB16000_OPC_UA_TRIGGER_ALARM".CLIENT.U2_STA3_COAXIAL.ALARMS.CAM_NO_LIGHT_DETECTED_A AND NOT "DB2120_MPP_ITC_IPC".RESET_FAULTS)) AND "DB7257_UNIT_2_STA_3_COAXIAL_ENABLE_DISABLE".ENABLED;
   "DB426_ALARMS_WARNINGS".ALARMS.UNIT_02.STATION_3_COAXIAL."720807" := "DB16000_OPC_UA_TRIGGER_ALARM".CLIENT.U2_STA3_COAXIAL.ALARMS.CAM_NO_LIGHT_DETECTED_A;
END_REGION

REGION Network 84: UNIT 2 STATION 3 COAXIAL CAMERA NO LASER DETECTED ALARM
   RUNG wire#powerrail
      { S7_Templates := "SrcType := Int" } EQ_Contact(in1 := "DB16005_U2_STA3_COAXIAL_CLIENT_INTERFACE".U2_STA3_CAM_Read.Variable.Status, in2 := -1)
      Contact( "DB16005_U2_STA3_COAXIAL_CLIENT_INTERFACE".U2_STA3_CAM_Read.Variable.NoLaserDetected )
      wire#w1
      Contact( "DB7257_UNIT_2_STA_3_COAXIAL_ENABLE_DISABLE".ENABLED )
      wire#w2
      Coil( "DB16000_OPC_UA_TRIGGER_ALARM".CLIENT.U2_STA3_COAXIAL.ALARMS.CAM_NO_LASER_DETECTED_A )
   END_RUNG
   RUNG wire#powerrail
      Contact( "DB16000_OPC_UA_TRIGGER_ALARM".CLIENT.U2_STA3_COAXIAL.ALARMS.CAM_NO_LASER_DETECTED_A )
      I_Contact( "DB2120_MPP_ITC_IPC".RESET_FAULTS )
   END_RUNG wire#w1
   RUNG wire#w2
      Coil( "DB426_ALARMS_WARNINGS".ALARMS.UNIT_02.STATION_3_COAXIAL."720808" )
   END_RUNG
   // the same network as SCL:
   "DB16000_OPC_UA_TRIGGER_ALARM".CLIENT.U2_STA3_COAXIAL.ALARMS.CAM_NO_LASER_DETECTED_A := ((("DB16005_U2_STA3_COAXIAL_CLIENT_INTERFACE".U2_STA3_CAM_Read.Variable.Status = (-1)) AND "DB16005_U2_STA3_COAXIAL_CLIENT_INTERFACE".U2_STA3_CAM_Read.Variable.NoLaserDetected) OR ("DB16000_OPC_UA_TRIGGER_ALARM".CLIENT.U2_STA3_COAXIAL.ALARMS.CAM_NO_LASER_DETECTED_A AND NOT "DB2120_MPP_ITC_IPC".RESET_FAULTS)) AND "DB7257_UNIT_2_STA_3_COAXIAL_ENABLE_DISABLE".ENABLED;
   "DB426_ALARMS_WARNINGS".ALARMS.UNIT_02.STATION_3_COAXIAL."720808" := "DB16000_OPC_UA_TRIGGER_ALARM".CLIENT.U2_STA3_COAXIAL.ALARMS.CAM_NO_LASER_DETECTED_A;
END_REGION

REGION Network 85: UNIT 2 STATION 3 COAXIAL CAMERA NO NOZZLE DETECTED ALARM
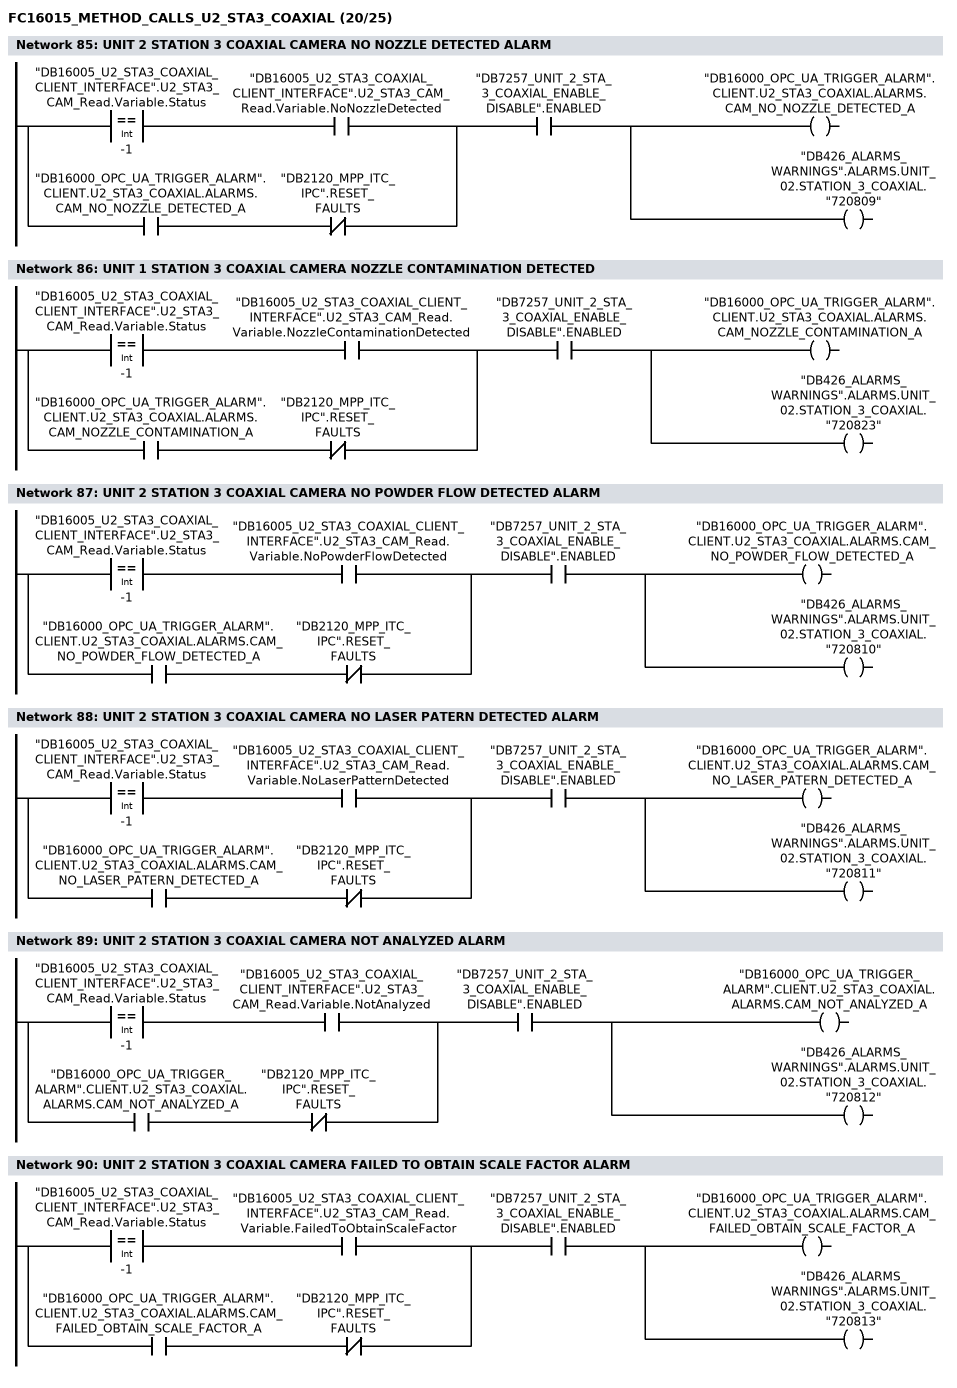
   RUNG wire#powerrail
      { S7_Templates := "SrcType := Int" } EQ_Contact(in1 := "DB16005_U2_STA3_COAXIAL_CLIENT_INTERFACE".U2_STA3_CAM_Read.Variable.Status, in2 := -1)
      Contact( "DB16005_U2_STA3_COAXIAL_CLIENT_INTERFACE".U2_STA3_CAM_Read.Variable.NoNozzleDetected )
      wire#w1
      Contact( "DB7257_UNIT_2_STA_3_COAXIAL_ENABLE_DISABLE".ENABLED )
      wire#w2
      Coil( "DB16000_OPC_UA_TRIGGER_ALARM".CLIENT.U2_STA3_COAXIAL.ALARMS.CAM_NO_NOZZLE_DETECTED_A )
   END_RUNG
   RUNG wire#powerrail
      Contact( "DB16000_OPC_UA_TRIGGER_ALARM".CLIENT.U2_STA3_COAXIAL.ALARMS.CAM_NO_NOZZLE_DETECTED_A )
      I_Contact( "DB2120_MPP_ITC_IPC".RESET_FAULTS )
   END_RUNG wire#w1
   RUNG wire#w2
      Coil( "DB426_ALARMS_WARNINGS".ALARMS.UNIT_02.STATION_3_COAXIAL."720809" )
   END_RUNG
   // the same network as SCL:
   "DB16000_OPC_UA_TRIGGER_ALARM".CLIENT.U2_STA3_COAXIAL.ALARMS.CAM_NO_NOZZLE_DETECTED_A := ((("DB16005_U2_STA3_COAXIAL_CLIENT_INTERFACE".U2_STA3_CAM_Read.Variable.Status = (-1)) AND "DB16005_U2_STA3_COAXIAL_CLIENT_INTERFACE".U2_STA3_CAM_Read.Variable.NoNozzleDetected) OR ("DB16000_OPC_UA_TRIGGER_ALARM".CLIENT.U2_STA3_COAXIAL.ALARMS.CAM_NO_NOZZLE_DETECTED_A AND NOT "DB2120_MPP_ITC_IPC".RESET_FAULTS)) AND "DB7257_UNIT_2_STA_3_COAXIAL_ENABLE_DISABLE".ENABLED;
   "DB426_ALARMS_WARNINGS".ALARMS.UNIT_02.STATION_3_COAXIAL."720809" := "DB16000_OPC_UA_TRIGGER_ALARM".CLIENT.U2_STA3_COAXIAL.ALARMS.CAM_NO_NOZZLE_DETECTED_A;
END_REGION

REGION Network 86: UNIT 1 STATION 3 COAXIAL CAMERA NOZZLE CONTAMINATION DETECTED
   RUNG wire#powerrail
      { S7_Templates := "SrcType := Int" } EQ_Contact(in1 := "DB16005_U2_STA3_COAXIAL_CLIENT_INTERFACE".U2_STA3_CAM_Read.Variable.Status, in2 := -1)
      Contact( "DB16005_U2_STA3_COAXIAL_CLIENT_INTERFACE".U2_STA3_CAM_Read.Variable.NozzleContaminationDetected )
      wire#w1
      Contact( "DB7257_UNIT_2_STA_3_COAXIAL_ENABLE_DISABLE".ENABLED )
      wire#w2
      Coil( "DB16000_OPC_UA_TRIGGER_ALARM".CLIENT.U2_STA3_COAXIAL.ALARMS.CAM_NOZZLE_CONTAMINATION_A )
   END_RUNG
   RUNG wire#powerrail
      Contact( "DB16000_OPC_UA_TRIGGER_ALARM".CLIENT.U2_STA3_COAXIAL.ALARMS.CAM_NOZZLE_CONTAMINATION_A )
      I_Contact( "DB2120_MPP_ITC_IPC".RESET_FAULTS )
   END_RUNG wire#w1
   RUNG wire#w2
      Coil( "DB426_ALARMS_WARNINGS".ALARMS.UNIT_02.STATION_3_COAXIAL."720823" )
   END_RUNG
   // the same network as SCL:
   "DB16000_OPC_UA_TRIGGER_ALARM".CLIENT.U2_STA3_COAXIAL.ALARMS.CAM_NOZZLE_CONTAMINATION_A := ((("DB16005_U2_STA3_COAXIAL_CLIENT_INTERFACE".U2_STA3_CAM_Read.Variable.Status = (-1)) AND "DB16005_U2_STA3_COAXIAL_CLIENT_INTERFACE".U2_STA3_CAM_Read.Variable.NozzleContaminationDetected) OR ("DB16000_OPC_UA_TRIGGER_ALARM".CLIENT.U2_STA3_COAXIAL.ALARMS.CAM_NOZZLE_CONTAMINATION_A AND NOT "DB2120_MPP_ITC_IPC".RESET_FAULTS)) AND "DB7257_UNIT_2_STA_3_COAXIAL_ENABLE_DISABLE".ENABLED;
   "DB426_ALARMS_WARNINGS".ALARMS.UNIT_02.STATION_3_COAXIAL."720823" := "DB16000_OPC_UA_TRIGGER_ALARM".CLIENT.U2_STA3_COAXIAL.ALARMS.CAM_NOZZLE_CONTAMINATION_A;
END_REGION

REGION Network 87: UNIT 2 STATION 3 COAXIAL CAMERA NO POWDER FLOW DETECTED ALARM
   RUNG wire#powerrail
      { S7_Templates := "SrcType := Int" } EQ_Contact(in1 := "DB16005_U2_STA3_COAXIAL_CLIENT_INTERFACE".U2_STA3_CAM_Read.Variable.Status, in2 := -1)
      Contact( "DB16005_U2_STA3_COAXIAL_CLIENT_INTERFACE".U2_STA3_CAM_Read.Variable.NoPowderFlowDetected )
      wire#w1
      Contact( "DB7257_UNIT_2_STA_3_COAXIAL_ENABLE_DISABLE".ENABLED )
      wire#w2
      Coil( "DB16000_OPC_UA_TRIGGER_ALARM".CLIENT.U2_STA3_COAXIAL.ALARMS.CAM_NO_POWDER_FLOW_DETECTED_A )
   END_RUNG
   RUNG wire#powerrail
      Contact( "DB16000_OPC_UA_TRIGGER_ALARM".CLIENT.U2_STA3_COAXIAL.ALARMS.CAM_NO_POWDER_FLOW_DETECTED_A )
      I_Contact( "DB2120_MPP_ITC_IPC".RESET_FAULTS )
   END_RUNG wire#w1
   RUNG wire#w2
      Coil( "DB426_ALARMS_WARNINGS".ALARMS.UNIT_02.STATION_3_COAXIAL."720810" )
   END_RUNG
   // the same network as SCL:
   "DB16000_OPC_UA_TRIGGER_ALARM".CLIENT.U2_STA3_COAXIAL.ALARMS.CAM_NO_POWDER_FLOW_DETECTED_A := ((("DB16005_U2_STA3_COAXIAL_CLIENT_INTERFACE".U2_STA3_CAM_Read.Variable.Status = (-1)) AND "DB16005_U2_STA3_COAXIAL_CLIENT_INTERFACE".U2_STA3_CAM_Read.Variable.NoPowderFlowDetected) OR ("DB16000_OPC_UA_TRIGGER_ALARM".CLIENT.U2_STA3_COAXIAL.ALARMS.CAM_NO_POWDER_FLOW_DETECTED_A AND NOT "DB2120_MPP_ITC_IPC".RESET_FAULTS)) AND "DB7257_UNIT_2_STA_3_COAXIAL_ENABLE_DISABLE".ENABLED;
   "DB426_ALARMS_WARNINGS".ALARMS.UNIT_02.STATION_3_COAXIAL."720810" := "DB16000_OPC_UA_TRIGGER_ALARM".CLIENT.U2_STA3_COAXIAL.ALARMS.CAM_NO_POWDER_FLOW_DETECTED_A;
END_REGION

REGION Network 88: UNIT 2 STATION 3 COAXIAL CAMERA NO LASER PATERN DETECTED ALARM
   RUNG wire#powerrail
      { S7_Templates := "SrcType := Int" } EQ_Contact(in1 := "DB16005_U2_STA3_COAXIAL_CLIENT_INTERFACE".U2_STA3_CAM_Read.Variable.Status, in2 := -1)
      Contact( "DB16005_U2_STA3_COAXIAL_CLIENT_INTERFACE".U2_STA3_CAM_Read.Variable.NoLaserPatternDetected )
      wire#w1
      Contact( "DB7257_UNIT_2_STA_3_COAXIAL_ENABLE_DISABLE".ENABLED )
      wire#w2
      Coil( "DB16000_OPC_UA_TRIGGER_ALARM".CLIENT.U2_STA3_COAXIAL.ALARMS.CAM_NO_LASER_PATERN_DETECTED_A )
   END_RUNG
   RUNG wire#powerrail
      Contact( "DB16000_OPC_UA_TRIGGER_ALARM".CLIENT.U2_STA3_COAXIAL.ALARMS.CAM_NO_LASER_PATERN_DETECTED_A )
      I_Contact( "DB2120_MPP_ITC_IPC".RESET_FAULTS )
   END_RUNG wire#w1
   RUNG wire#w2
      Coil( "DB426_ALARMS_WARNINGS".ALARMS.UNIT_02.STATION_3_COAXIAL."720811" )
   END_RUNG
   // the same network as SCL:
   "DB16000_OPC_UA_TRIGGER_ALARM".CLIENT.U2_STA3_COAXIAL.ALARMS.CAM_NO_LASER_PATERN_DETECTED_A := ((("DB16005_U2_STA3_COAXIAL_CLIENT_INTERFACE".U2_STA3_CAM_Read.Variable.Status = (-1)) AND "DB16005_U2_STA3_COAXIAL_CLIENT_INTERFACE".U2_STA3_CAM_Read.Variable.NoLaserPatternDetected) OR ("DB16000_OPC_UA_TRIGGER_ALARM".CLIENT.U2_STA3_COAXIAL.ALARMS.CAM_NO_LASER_PATERN_DETECTED_A AND NOT "DB2120_MPP_ITC_IPC".RESET_FAULTS)) AND "DB7257_UNIT_2_STA_3_COAXIAL_ENABLE_DISABLE".ENABLED;
   "DB426_ALARMS_WARNINGS".ALARMS.UNIT_02.STATION_3_COAXIAL."720811" := "DB16000_OPC_UA_TRIGGER_ALARM".CLIENT.U2_STA3_COAXIAL.ALARMS.CAM_NO_LASER_PATERN_DETECTED_A;
END_REGION

REGION Network 89: UNIT 2 STATION 3 COAXIAL CAMERA NOT ANALYZED ALARM
   RUNG wire#powerrail
      { S7_Templates := "SrcType := Int" } EQ_Contact(in1 := "DB16005_U2_STA3_COAXIAL_CLIENT_INTERFACE".U2_STA3_CAM_Read.Variable.Status, in2 := -1)
      Contact( "DB16005_U2_STA3_COAXIAL_CLIENT_INTERFACE".U2_STA3_CAM_Read.Variable.NotAnalyzed )
      wire#w1
      Contact( "DB7257_UNIT_2_STA_3_COAXIAL_ENABLE_DISABLE".ENABLED )
      wire#w2
      Coil( "DB16000_OPC_UA_TRIGGER_ALARM".CLIENT.U2_STA3_COAXIAL.ALARMS.CAM_NOT_ANALYZED_A )
   END_RUNG
   RUNG wire#powerrail
      Contact( "DB16000_OPC_UA_TRIGGER_ALARM".CLIENT.U2_STA3_COAXIAL.ALARMS.CAM_NOT_ANALYZED_A )
      I_Contact( "DB2120_MPP_ITC_IPC".RESET_FAULTS )
   END_RUNG wire#w1
   RUNG wire#w2
      Coil( "DB426_ALARMS_WARNINGS".ALARMS.UNIT_02.STATION_3_COAXIAL."720812" )
   END_RUNG
   // the same network as SCL:
   "DB16000_OPC_UA_TRIGGER_ALARM".CLIENT.U2_STA3_COAXIAL.ALARMS.CAM_NOT_ANALYZED_A := ((("DB16005_U2_STA3_COAXIAL_CLIENT_INTERFACE".U2_STA3_CAM_Read.Variable.Status = (-1)) AND "DB16005_U2_STA3_COAXIAL_CLIENT_INTERFACE".U2_STA3_CAM_Read.Variable.NotAnalyzed) OR ("DB16000_OPC_UA_TRIGGER_ALARM".CLIENT.U2_STA3_COAXIAL.ALARMS.CAM_NOT_ANALYZED_A AND NOT "DB2120_MPP_ITC_IPC".RESET_FAULTS)) AND "DB7257_UNIT_2_STA_3_COAXIAL_ENABLE_DISABLE".ENABLED;
   "DB426_ALARMS_WARNINGS".ALARMS.UNIT_02.STATION_3_COAXIAL."720812" := "DB16000_OPC_UA_TRIGGER_ALARM".CLIENT.U2_STA3_COAXIAL.ALARMS.CAM_NOT_ANALYZED_A;
END_REGION

REGION Network 90: UNIT 2 STATION 3 COAXIAL CAMERA FAILED TO OBTAIN SCALE FACTOR ALARM
   RUNG wire#powerrail
      { S7_Templates := "SrcType := Int" } EQ_Contact(in1 := "DB16005_U2_STA3_COAXIAL_CLIENT_INTERFACE".U2_STA3_CAM_Read.Variable.Status, in2 := -1)
      Contact( "DB16005_U2_STA3_COAXIAL_CLIENT_INTERFACE".U2_STA3_CAM_Read.Variable.FailedToObtainScaleFactor )
      wire#w1
      Contact( "DB7257_UNIT_2_STA_3_COAXIAL_ENABLE_DISABLE".ENABLED )
      wire#w2
      Coil( "DB16000_OPC_UA_TRIGGER_ALARM".CLIENT.U2_STA3_COAXIAL.ALARMS.CAM_FAILED_OBTAIN_SCALE_FACTOR_A )
   END_RUNG
   RUNG wire#powerrail
      Contact( "DB16000_OPC_UA_TRIGGER_ALARM".CLIENT.U2_STA3_COAXIAL.ALARMS.CAM_FAILED_OBTAIN_SCALE_FACTOR_A )
      I_Contact( "DB2120_MPP_ITC_IPC".RESET_FAULTS )
   END_RUNG wire#w1
   RUNG wire#w2
      Coil( "DB426_ALARMS_WARNINGS".ALARMS.UNIT_02.STATION_3_COAXIAL."720813" )
   END_RUNG
   // the same network as SCL:
   "DB16000_OPC_UA_TRIGGER_ALARM".CLIENT.U2_STA3_COAXIAL.ALARMS.CAM_FAILED_OBTAIN_SCALE_FACTOR_A := ((("DB16005_U2_STA3_COAXIAL_CLIENT_INTERFACE".U2_STA3_CAM_Read.Variable.Status = (-1)) AND "DB16005_U2_STA3_COAXIAL_CLIENT_INTERFACE".U2_STA3_CAM_Read.Variable.FailedToObtainScaleFactor) OR ("DB16000_OPC_UA_TRIGGER_ALARM".CLIENT.U2_STA3_COAXIAL.ALARMS.CAM_FAILED_OBTAIN_SCALE_FACTOR_A AND NOT "DB2120_MPP_ITC_IPC".RESET_FAULTS)) AND "DB7257_UNIT_2_STA_3_COAXIAL_ENABLE_DISABLE".ENABLED;
   "DB426_ALARMS_WARNINGS".ALARMS.UNIT_02.STATION_3_COAXIAL."720813" := "DB16000_OPC_UA_TRIGGER_ALARM".CLIENT.U2_STA3_COAXIAL.ALARMS.CAM_FAILED_OBTAIN_SCALE_FACTOR_A;
END_REGION

REGION Network 91: UNIT 2 STATION 3 COAXIAL CAMERA UNALIGNED POWDER FLOW VORTEX ALARM
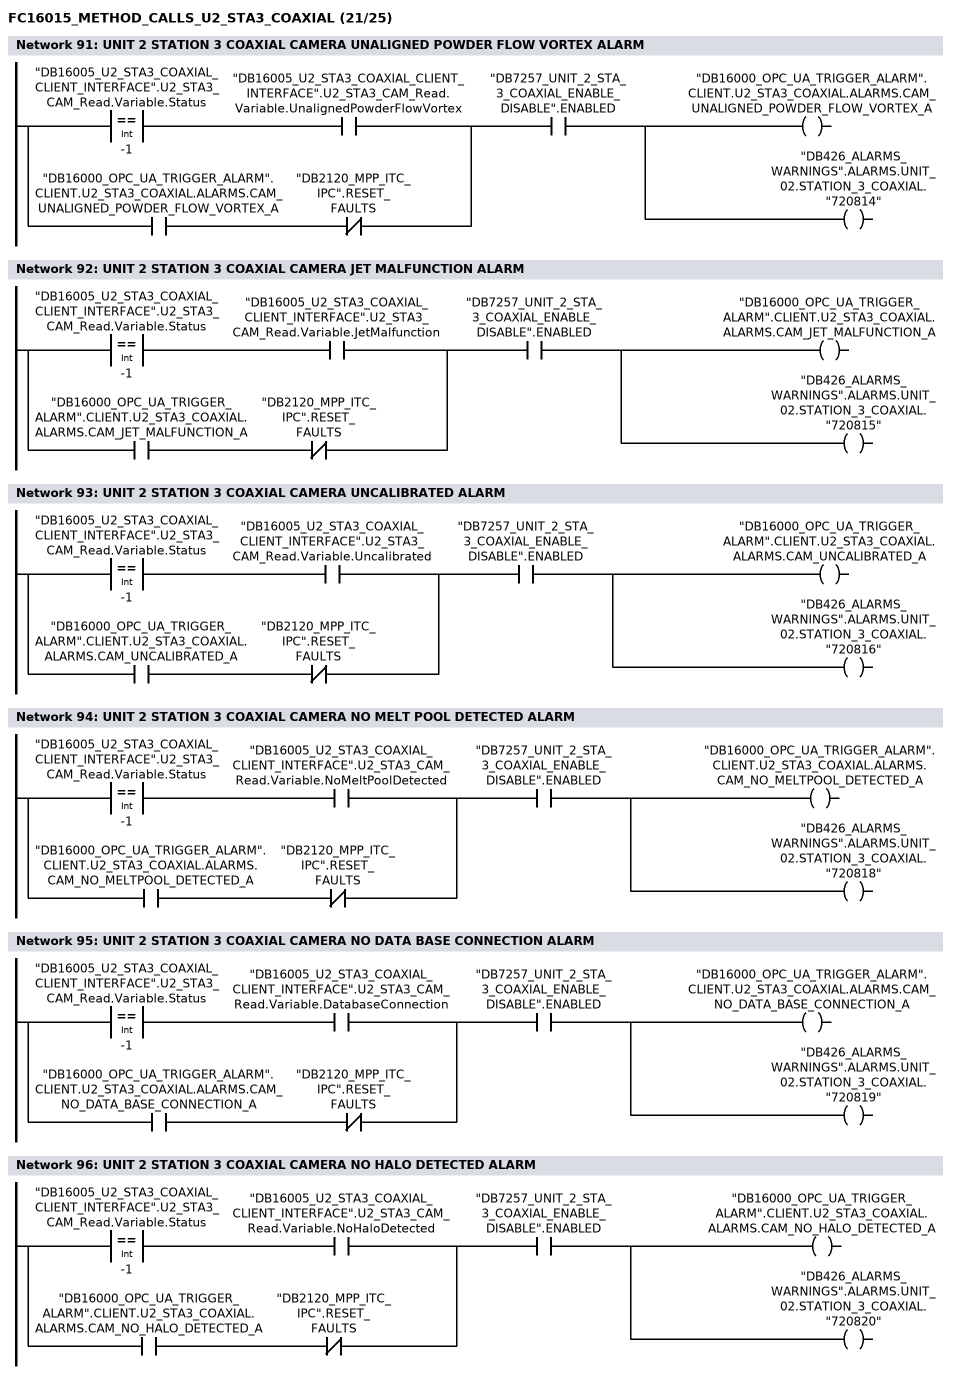
   RUNG wire#powerrail
      { S7_Templates := "SrcType := Int" } EQ_Contact(in1 := "DB16005_U2_STA3_COAXIAL_CLIENT_INTERFACE".U2_STA3_CAM_Read.Variable.Status, in2 := -1)
      Contact( "DB16005_U2_STA3_COAXIAL_CLIENT_INTERFACE".U2_STA3_CAM_Read.Variable.UnalignedPowderFlowVortex )
      wire#w1
      Contact( "DB7257_UNIT_2_STA_3_COAXIAL_ENABLE_DISABLE".ENABLED )
      wire#w2
      Coil( "DB16000_OPC_UA_TRIGGER_ALARM".CLIENT.U2_STA3_COAXIAL.ALARMS.CAM_UNALIGNED_POWDER_FLOW_VORTEX_A )
   END_RUNG
   RUNG wire#powerrail
      Contact( "DB16000_OPC_UA_TRIGGER_ALARM".CLIENT.U2_STA3_COAXIAL.ALARMS.CAM_UNALIGNED_POWDER_FLOW_VORTEX_A )
      I_Contact( "DB2120_MPP_ITC_IPC".RESET_FAULTS )
   END_RUNG wire#w1
   RUNG wire#w2
      Coil( "DB426_ALARMS_WARNINGS".ALARMS.UNIT_02.STATION_3_COAXIAL."720814" )
   END_RUNG
   // the same network as SCL:
   "DB16000_OPC_UA_TRIGGER_ALARM".CLIENT.U2_STA3_COAXIAL.ALARMS.CAM_UNALIGNED_POWDER_FLOW_VORTEX_A := ((("DB16005_U2_STA3_COAXIAL_CLIENT_INTERFACE".U2_STA3_CAM_Read.Variable.Status = (-1)) AND "DB16005_U2_STA3_COAXIAL_CLIENT_INTERFACE".U2_STA3_CAM_Read.Variable.UnalignedPowderFlowVortex) OR ("DB16000_OPC_UA_TRIGGER_ALARM".CLIENT.U2_STA3_COAXIAL.ALARMS.CAM_UNALIGNED_POWDER_FLOW_VORTEX_A AND NOT "DB2120_MPP_ITC_IPC".RESET_FAULTS)) AND "DB7257_UNIT_2_STA_3_COAXIAL_ENABLE_DISABLE".ENABLED;
   "DB426_ALARMS_WARNINGS".ALARMS.UNIT_02.STATION_3_COAXIAL."720814" := "DB16000_OPC_UA_TRIGGER_ALARM".CLIENT.U2_STA3_COAXIAL.ALARMS.CAM_UNALIGNED_POWDER_FLOW_VORTEX_A;
END_REGION

REGION Network 92: UNIT 2 STATION 3 COAXIAL CAMERA JET MALFUNCTION ALARM
   RUNG wire#powerrail
      { S7_Templates := "SrcType := Int" } EQ_Contact(in1 := "DB16005_U2_STA3_COAXIAL_CLIENT_INTERFACE".U2_STA3_CAM_Read.Variable.Status, in2 := -1)
      Contact( "DB16005_U2_STA3_COAXIAL_CLIENT_INTERFACE".U2_STA3_CAM_Read.Variable.JetMalfunction )
      wire#w1
      Contact( "DB7257_UNIT_2_STA_3_COAXIAL_ENABLE_DISABLE".ENABLED )
      wire#w2
      Coil( "DB16000_OPC_UA_TRIGGER_ALARM".CLIENT.U2_STA3_COAXIAL.ALARMS.CAM_JET_MALFUNCTION_A )
   END_RUNG
   RUNG wire#powerrail
      Contact( "DB16000_OPC_UA_TRIGGER_ALARM".CLIENT.U2_STA3_COAXIAL.ALARMS.CAM_JET_MALFUNCTION_A )
      I_Contact( "DB2120_MPP_ITC_IPC".RESET_FAULTS )
   END_RUNG wire#w1
   RUNG wire#w2
      Coil( "DB426_ALARMS_WARNINGS".ALARMS.UNIT_02.STATION_3_COAXIAL."720815" )
   END_RUNG
   // the same network as SCL:
   "DB16000_OPC_UA_TRIGGER_ALARM".CLIENT.U2_STA3_COAXIAL.ALARMS.CAM_JET_MALFUNCTION_A := ((("DB16005_U2_STA3_COAXIAL_CLIENT_INTERFACE".U2_STA3_CAM_Read.Variable.Status = (-1)) AND "DB16005_U2_STA3_COAXIAL_CLIENT_INTERFACE".U2_STA3_CAM_Read.Variable.JetMalfunction) OR ("DB16000_OPC_UA_TRIGGER_ALARM".CLIENT.U2_STA3_COAXIAL.ALARMS.CAM_JET_MALFUNCTION_A AND NOT "DB2120_MPP_ITC_IPC".RESET_FAULTS)) AND "DB7257_UNIT_2_STA_3_COAXIAL_ENABLE_DISABLE".ENABLED;
   "DB426_ALARMS_WARNINGS".ALARMS.UNIT_02.STATION_3_COAXIAL."720815" := "DB16000_OPC_UA_TRIGGER_ALARM".CLIENT.U2_STA3_COAXIAL.ALARMS.CAM_JET_MALFUNCTION_A;
END_REGION

REGION Network 93: UNIT 2 STATION 3 COAXIAL CAMERA UNCALIBRATED ALARM
   RUNG wire#powerrail
      { S7_Templates := "SrcType := Int" } EQ_Contact(in1 := "DB16005_U2_STA3_COAXIAL_CLIENT_INTERFACE".U2_STA3_CAM_Read.Variable.Status, in2 := -1)
      Contact( "DB16005_U2_STA3_COAXIAL_CLIENT_INTERFACE".U2_STA3_CAM_Read.Variable.Uncalibrated )
      wire#w1
      Contact( "DB7257_UNIT_2_STA_3_COAXIAL_ENABLE_DISABLE".ENABLED )
      wire#w2
      Coil( "DB16000_OPC_UA_TRIGGER_ALARM".CLIENT.U2_STA3_COAXIAL.ALARMS.CAM_UNCALIBRATED_A )
   END_RUNG
   RUNG wire#powerrail
      Contact( "DB16000_OPC_UA_TRIGGER_ALARM".CLIENT.U2_STA3_COAXIAL.ALARMS.CAM_UNCALIBRATED_A )
      I_Contact( "DB2120_MPP_ITC_IPC".RESET_FAULTS )
   END_RUNG wire#w1
   RUNG wire#w2
      Coil( "DB426_ALARMS_WARNINGS".ALARMS.UNIT_02.STATION_3_COAXIAL."720816" )
   END_RUNG
   // the same network as SCL:
   "DB16000_OPC_UA_TRIGGER_ALARM".CLIENT.U2_STA3_COAXIAL.ALARMS.CAM_UNCALIBRATED_A := ((("DB16005_U2_STA3_COAXIAL_CLIENT_INTERFACE".U2_STA3_CAM_Read.Variable.Status = (-1)) AND "DB16005_U2_STA3_COAXIAL_CLIENT_INTERFACE".U2_STA3_CAM_Read.Variable.Uncalibrated) OR ("DB16000_OPC_UA_TRIGGER_ALARM".CLIENT.U2_STA3_COAXIAL.ALARMS.CAM_UNCALIBRATED_A AND NOT "DB2120_MPP_ITC_IPC".RESET_FAULTS)) AND "DB7257_UNIT_2_STA_3_COAXIAL_ENABLE_DISABLE".ENABLED;
   "DB426_ALARMS_WARNINGS".ALARMS.UNIT_02.STATION_3_COAXIAL."720816" := "DB16000_OPC_UA_TRIGGER_ALARM".CLIENT.U2_STA3_COAXIAL.ALARMS.CAM_UNCALIBRATED_A;
END_REGION

REGION Network 94: UNIT 2 STATION 3 COAXIAL CAMERA NO MELT POOL DETECTED ALARM
   RUNG wire#powerrail
      { S7_Templates := "SrcType := Int" } EQ_Contact(in1 := "DB16005_U2_STA3_COAXIAL_CLIENT_INTERFACE".U2_STA3_CAM_Read.Variable.Status, in2 := -1)
      Contact( "DB16005_U2_STA3_COAXIAL_CLIENT_INTERFACE".U2_STA3_CAM_Read.Variable.NoMeltPoolDetected )
      wire#w1
      Contact( "DB7257_UNIT_2_STA_3_COAXIAL_ENABLE_DISABLE".ENABLED )
      wire#w2
      Coil( "DB16000_OPC_UA_TRIGGER_ALARM".CLIENT.U2_STA3_COAXIAL.ALARMS.CAM_NO_MELTPOOL_DETECTED_A )
   END_RUNG
   RUNG wire#powerrail
      Contact( "DB16000_OPC_UA_TRIGGER_ALARM".CLIENT.U2_STA3_COAXIAL.ALARMS.CAM_NO_MELTPOOL_DETECTED_A )
      I_Contact( "DB2120_MPP_ITC_IPC".RESET_FAULTS )
   END_RUNG wire#w1
   RUNG wire#w2
      Coil( "DB426_ALARMS_WARNINGS".ALARMS.UNIT_02.STATION_3_COAXIAL."720818" )
   END_RUNG
   // the same network as SCL:
   "DB16000_OPC_UA_TRIGGER_ALARM".CLIENT.U2_STA3_COAXIAL.ALARMS.CAM_NO_MELTPOOL_DETECTED_A := ((("DB16005_U2_STA3_COAXIAL_CLIENT_INTERFACE".U2_STA3_CAM_Read.Variable.Status = (-1)) AND "DB16005_U2_STA3_COAXIAL_CLIENT_INTERFACE".U2_STA3_CAM_Read.Variable.NoMeltPoolDetected) OR ("DB16000_OPC_UA_TRIGGER_ALARM".CLIENT.U2_STA3_COAXIAL.ALARMS.CAM_NO_MELTPOOL_DETECTED_A AND NOT "DB2120_MPP_ITC_IPC".RESET_FAULTS)) AND "DB7257_UNIT_2_STA_3_COAXIAL_ENABLE_DISABLE".ENABLED;
   "DB426_ALARMS_WARNINGS".ALARMS.UNIT_02.STATION_3_COAXIAL."720818" := "DB16000_OPC_UA_TRIGGER_ALARM".CLIENT.U2_STA3_COAXIAL.ALARMS.CAM_NO_MELTPOOL_DETECTED_A;
END_REGION

REGION Network 95: UNIT 2 STATION 3 COAXIAL CAMERA NO DATA BASE CONNECTION ALARM
   RUNG wire#powerrail
      { S7_Templates := "SrcType := Int" } EQ_Contact(in1 := "DB16005_U2_STA3_COAXIAL_CLIENT_INTERFACE".U2_STA3_CAM_Read.Variable.Status, in2 := -1)
      Contact( "DB16005_U2_STA3_COAXIAL_CLIENT_INTERFACE".U2_STA3_CAM_Read.Variable.DatabaseConnection )
      wire#w1
      Contact( "DB7257_UNIT_2_STA_3_COAXIAL_ENABLE_DISABLE".ENABLED )
      wire#w2
      Coil( "DB16000_OPC_UA_TRIGGER_ALARM".CLIENT.U2_STA3_COAXIAL.ALARMS.CAM_NO_DATA_BASE_CONNECTION_A )
   END_RUNG
   RUNG wire#powerrail
      Contact( "DB16000_OPC_UA_TRIGGER_ALARM".CLIENT.U2_STA3_COAXIAL.ALARMS.CAM_NO_DATA_BASE_CONNECTION_A )
      I_Contact( "DB2120_MPP_ITC_IPC".RESET_FAULTS )
   END_RUNG wire#w1
   RUNG wire#w2
      Coil( "DB426_ALARMS_WARNINGS".ALARMS.UNIT_02.STATION_3_COAXIAL."720819" )
   END_RUNG
   // the same network as SCL:
   "DB16000_OPC_UA_TRIGGER_ALARM".CLIENT.U2_STA3_COAXIAL.ALARMS.CAM_NO_DATA_BASE_CONNECTION_A := ((("DB16005_U2_STA3_COAXIAL_CLIENT_INTERFACE".U2_STA3_CAM_Read.Variable.Status = (-1)) AND "DB16005_U2_STA3_COAXIAL_CLIENT_INTERFACE".U2_STA3_CAM_Read.Variable.DatabaseConnection) OR ("DB16000_OPC_UA_TRIGGER_ALARM".CLIENT.U2_STA3_COAXIAL.ALARMS.CAM_NO_DATA_BASE_CONNECTION_A AND NOT "DB2120_MPP_ITC_IPC".RESET_FAULTS)) AND "DB7257_UNIT_2_STA_3_COAXIAL_ENABLE_DISABLE".ENABLED;
   "DB426_ALARMS_WARNINGS".ALARMS.UNIT_02.STATION_3_COAXIAL."720819" := "DB16000_OPC_UA_TRIGGER_ALARM".CLIENT.U2_STA3_COAXIAL.ALARMS.CAM_NO_DATA_BASE_CONNECTION_A;
END_REGION

REGION Network 96: UNIT 2 STATION 3 COAXIAL CAMERA NO HALO DETECTED ALARM
   RUNG wire#powerrail
      { S7_Templates := "SrcType := Int" } EQ_Contact(in1 := "DB16005_U2_STA3_COAXIAL_CLIENT_INTERFACE".U2_STA3_CAM_Read.Variable.Status, in2 := -1)
      Contact( "DB16005_U2_STA3_COAXIAL_CLIENT_INTERFACE".U2_STA3_CAM_Read.Variable.NoHaloDetected )
      wire#w1
      Contact( "DB7257_UNIT_2_STA_3_COAXIAL_ENABLE_DISABLE".ENABLED )
      wire#w2
      Coil( "DB16000_OPC_UA_TRIGGER_ALARM".CLIENT.U2_STA3_COAXIAL.ALARMS.CAM_NO_HALO_DETECTED_A )
   END_RUNG
   RUNG wire#powerrail
      Contact( "DB16000_OPC_UA_TRIGGER_ALARM".CLIENT.U2_STA3_COAXIAL.ALARMS.CAM_NO_HALO_DETECTED_A )
      I_Contact( "DB2120_MPP_ITC_IPC".RESET_FAULTS )
   END_RUNG wire#w1
   RUNG wire#w2
      Coil( "DB426_ALARMS_WARNINGS".ALARMS.UNIT_02.STATION_3_COAXIAL."720820" )
   END_RUNG
   // the same network as SCL:
   "DB16000_OPC_UA_TRIGGER_ALARM".CLIENT.U2_STA3_COAXIAL.ALARMS.CAM_NO_HALO_DETECTED_A := ((("DB16005_U2_STA3_COAXIAL_CLIENT_INTERFACE".U2_STA3_CAM_Read.Variable.Status = (-1)) AND "DB16005_U2_STA3_COAXIAL_CLIENT_INTERFACE".U2_STA3_CAM_Read.Variable.NoHaloDetected) OR ("DB16000_OPC_UA_TRIGGER_ALARM".CLIENT.U2_STA3_COAXIAL.ALARMS.CAM_NO_HALO_DETECTED_A AND NOT "DB2120_MPP_ITC_IPC".RESET_FAULTS)) AND "DB7257_UNIT_2_STA_3_COAXIAL_ENABLE_DISABLE".ENABLED;
   "DB426_ALARMS_WARNINGS".ALARMS.UNIT_02.STATION_3_COAXIAL."720820" := "DB16000_OPC_UA_TRIGGER_ALARM".CLIENT.U2_STA3_COAXIAL.ALARMS.CAM_NO_HALO_DETECTED_A;
END_REGION

REGION Network 97: UNIT 2 STATION 3 COAXIAL CAMERA STORAGE ERROR ALARM
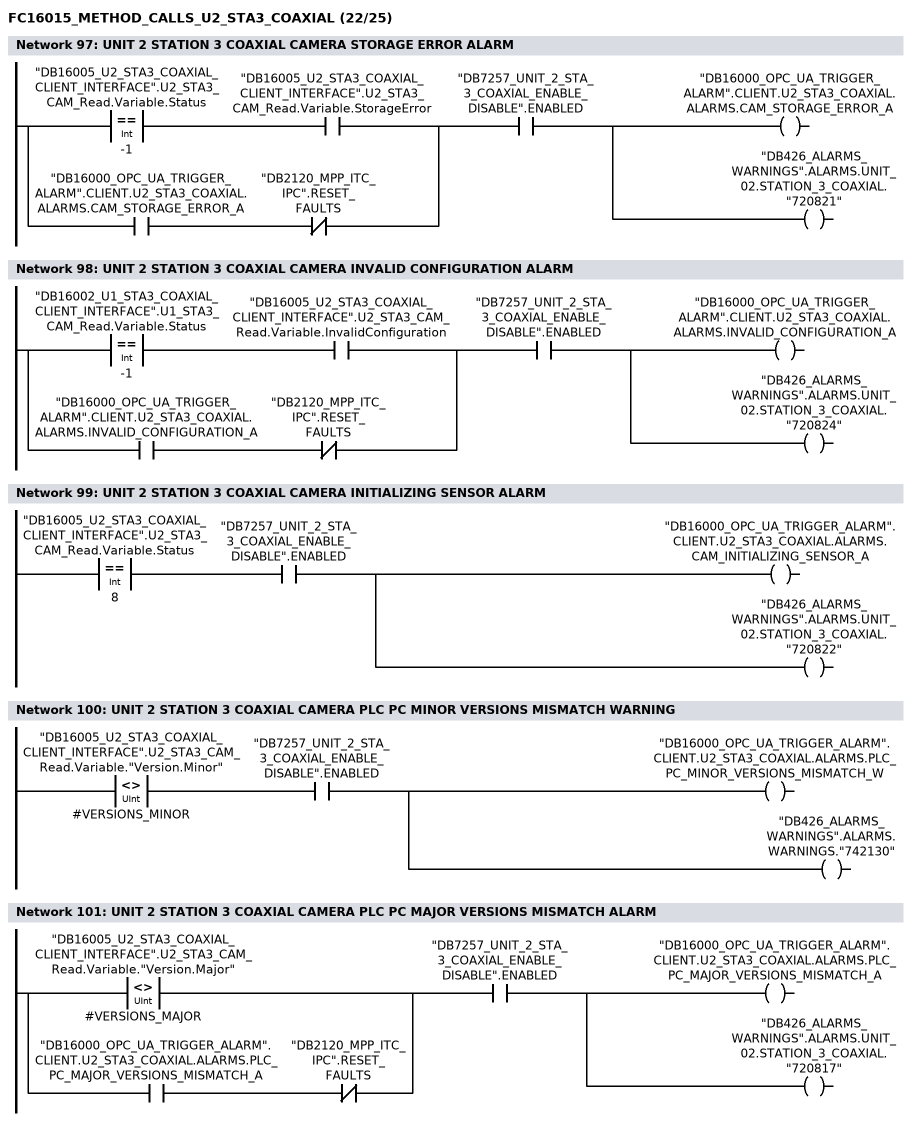
   RUNG wire#powerrail
      { S7_Templates := "SrcType := Int" } EQ_Contact(in1 := "DB16005_U2_STA3_COAXIAL_CLIENT_INTERFACE".U2_STA3_CAM_Read.Variable.Status, in2 := -1)
      Contact( "DB16005_U2_STA3_COAXIAL_CLIENT_INTERFACE".U2_STA3_CAM_Read.Variable.StorageError )
      wire#w1
      Contact( "DB7257_UNIT_2_STA_3_COAXIAL_ENABLE_DISABLE".ENABLED )
      wire#w2
      Coil( "DB16000_OPC_UA_TRIGGER_ALARM".CLIENT.U2_STA3_COAXIAL.ALARMS.CAM_STORAGE_ERROR_A )
   END_RUNG
   RUNG wire#powerrail
      Contact( "DB16000_OPC_UA_TRIGGER_ALARM".CLIENT.U2_STA3_COAXIAL.ALARMS.CAM_STORAGE_ERROR_A )
      I_Contact( "DB2120_MPP_ITC_IPC".RESET_FAULTS )
   END_RUNG wire#w1
   RUNG wire#w2
      Coil( "DB426_ALARMS_WARNINGS".ALARMS.UNIT_02.STATION_3_COAXIAL."720821" )
   END_RUNG
   // the same network as SCL:
   "DB16000_OPC_UA_TRIGGER_ALARM".CLIENT.U2_STA3_COAXIAL.ALARMS.CAM_STORAGE_ERROR_A := ((("DB16005_U2_STA3_COAXIAL_CLIENT_INTERFACE".U2_STA3_CAM_Read.Variable.Status = (-1)) AND "DB16005_U2_STA3_COAXIAL_CLIENT_INTERFACE".U2_STA3_CAM_Read.Variable.StorageError) OR ("DB16000_OPC_UA_TRIGGER_ALARM".CLIENT.U2_STA3_COAXIAL.ALARMS.CAM_STORAGE_ERROR_A AND NOT "DB2120_MPP_ITC_IPC".RESET_FAULTS)) AND "DB7257_UNIT_2_STA_3_COAXIAL_ENABLE_DISABLE".ENABLED;
   "DB426_ALARMS_WARNINGS".ALARMS.UNIT_02.STATION_3_COAXIAL."720821" := "DB16000_OPC_UA_TRIGGER_ALARM".CLIENT.U2_STA3_COAXIAL.ALARMS.CAM_STORAGE_ERROR_A;
END_REGION

REGION Network 98: UNIT 2 STATION 3 COAXIAL CAMERA INVALID CONFIGURATION ALARM
   RUNG wire#powerrail
      { S7_Templates := "SrcType := Int" } EQ_Contact(in1 := "DB16002_U1_STA3_COAXIAL_CLIENT_INTERFACE".U1_STA3_CAM_Read.Variable.Status, in2 := -1)
      Contact( "DB16005_U2_STA3_COAXIAL_CLIENT_INTERFACE".U2_STA3_CAM_Read.Variable.InvalidConfiguration )
      wire#w1
      Contact( "DB7257_UNIT_2_STA_3_COAXIAL_ENABLE_DISABLE".ENABLED )
      wire#w2
      Coil( "DB16000_OPC_UA_TRIGGER_ALARM".CLIENT.U2_STA3_COAXIAL.ALARMS.INVALID_CONFIGURATION_A )
   END_RUNG
   RUNG wire#powerrail
      Contact( "DB16000_OPC_UA_TRIGGER_ALARM".CLIENT.U2_STA3_COAXIAL.ALARMS.INVALID_CONFIGURATION_A )
      I_Contact( "DB2120_MPP_ITC_IPC".RESET_FAULTS )
   END_RUNG wire#w1
   RUNG wire#w2
      Coil( "DB426_ALARMS_WARNINGS".ALARMS.UNIT_02.STATION_3_COAXIAL."720824" )
   END_RUNG
   // the same network as SCL:
   "DB16000_OPC_UA_TRIGGER_ALARM".CLIENT.U2_STA3_COAXIAL.ALARMS.INVALID_CONFIGURATION_A := ((("DB16002_U1_STA3_COAXIAL_CLIENT_INTERFACE".U1_STA3_CAM_Read.Variable.Status = (-1)) AND "DB16005_U2_STA3_COAXIAL_CLIENT_INTERFACE".U2_STA3_CAM_Read.Variable.InvalidConfiguration) OR ("DB16000_OPC_UA_TRIGGER_ALARM".CLIENT.U2_STA3_COAXIAL.ALARMS.INVALID_CONFIGURATION_A AND NOT "DB2120_MPP_ITC_IPC".RESET_FAULTS)) AND "DB7257_UNIT_2_STA_3_COAXIAL_ENABLE_DISABLE".ENABLED;
   "DB426_ALARMS_WARNINGS".ALARMS.UNIT_02.STATION_3_COAXIAL."720824" := "DB16000_OPC_UA_TRIGGER_ALARM".CLIENT.U2_STA3_COAXIAL.ALARMS.INVALID_CONFIGURATION_A;
END_REGION

REGION Network 99: UNIT 2 STATION 3 COAXIAL CAMERA INITIALIZING SENSOR ALARM
   RUNG wire#powerrail
      { S7_Templates := "SrcType := Int" } EQ_Contact(in1 := "DB16005_U2_STA3_COAXIAL_CLIENT_INTERFACE".U2_STA3_CAM_Read.Variable.Status, in2 := 8)
      Contact( "DB7257_UNIT_2_STA_3_COAXIAL_ENABLE_DISABLE".ENABLED )
      wire#w1
      Coil( "DB16000_OPC_UA_TRIGGER_ALARM".CLIENT.U2_STA3_COAXIAL.ALARMS.CAM_INITIALIZING_SENSOR_A )
   END_RUNG
   RUNG wire#w1
      Coil( "DB426_ALARMS_WARNINGS".ALARMS.UNIT_02.STATION_3_COAXIAL."720822" )
   END_RUNG
   // the same network as SCL:
   "DB16000_OPC_UA_TRIGGER_ALARM".CLIENT.U2_STA3_COAXIAL.ALARMS.CAM_INITIALIZING_SENSOR_A := ("DB16005_U2_STA3_COAXIAL_CLIENT_INTERFACE".U2_STA3_CAM_Read.Variable.Status = 8) AND "DB7257_UNIT_2_STA_3_COAXIAL_ENABLE_DISABLE".ENABLED;
   "DB426_ALARMS_WARNINGS".ALARMS.UNIT_02.STATION_3_COAXIAL."720822" := "DB16000_OPC_UA_TRIGGER_ALARM".CLIENT.U2_STA3_COAXIAL.ALARMS.CAM_INITIALIZING_SENSOR_A;
END_REGION

REGION Network 100: UNIT 2 STATION 3 COAXIAL CAMERA PLC PC MINOR VERSIONS MISMATCH WARNING
   RUNG wire#powerrail
      { S7_Templates := "SrcType := UInt" } NE_Contact(in1 := "DB16005_U2_STA3_COAXIAL_CLIENT_INTERFACE".U2_STA3_CAM_Read.Variable."Version.Minor", in2 := #VERSIONS_MINOR)
      Contact( "DB7257_UNIT_2_STA_3_COAXIAL_ENABLE_DISABLE".ENABLED )
      wire#w1
      Coil( "DB16000_OPC_UA_TRIGGER_ALARM".CLIENT.U2_STA3_COAXIAL.ALARMS.PLC_PC_MINOR_VERSIONS_MISMATCH_W )
   END_RUNG
   RUNG wire#w1
      Coil( "DB426_ALARMS_WARNINGS".ALARMS.WARNINGS."742130" )
   END_RUNG
   // the same network as SCL:
   "DB16000_OPC_UA_TRIGGER_ALARM".CLIENT.U2_STA3_COAXIAL.ALARMS.PLC_PC_MINOR_VERSIONS_MISMATCH_W := ("DB16005_U2_STA3_COAXIAL_CLIENT_INTERFACE".U2_STA3_CAM_Read.Variable."Version.Minor" <> #VERSIONS_MINOR) AND "DB7257_UNIT_2_STA_3_COAXIAL_ENABLE_DISABLE".ENABLED;
   "DB426_ALARMS_WARNINGS".ALARMS.WARNINGS."742130" := "DB16000_OPC_UA_TRIGGER_ALARM".CLIENT.U2_STA3_COAXIAL.ALARMS.PLC_PC_MINOR_VERSIONS_MISMATCH_W;
END_REGION

REGION Network 101: UNIT 2 STATION 3 COAXIAL CAMERA PLC PC MAJOR VERSIONS MISMATCH ALARM
   RUNG wire#powerrail
      { S7_Templates := "SrcType := UInt" } NE_Contact(in1 := "DB16005_U2_STA3_COAXIAL_CLIENT_INTERFACE".U2_STA3_CAM_Read.Variable."Version.Major", in2 := #VERSIONS_MAJOR)
      wire#w1
      Contact( "DB7257_UNIT_2_STA_3_COAXIAL_ENABLE_DISABLE".ENABLED )
      wire#w2
      Coil( "DB16000_OPC_UA_TRIGGER_ALARM".CLIENT.U2_STA3_COAXIAL.ALARMS.PLC_PC_MAJOR_VERSIONS_MISMATCH_A )
   END_RUNG
   RUNG wire#powerrail
      Contact( "DB16000_OPC_UA_TRIGGER_ALARM".CLIENT.U2_STA3_COAXIAL.ALARMS.PLC_PC_MAJOR_VERSIONS_MISMATCH_A )
      I_Contact( "DB2120_MPP_ITC_IPC".RESET_FAULTS )
   END_RUNG wire#w1
   RUNG wire#w2
      Coil( "DB426_ALARMS_WARNINGS".ALARMS.UNIT_02.STATION_3_COAXIAL."720817" )
   END_RUNG
   // the same network as SCL:
   "DB16000_OPC_UA_TRIGGER_ALARM".CLIENT.U2_STA3_COAXIAL.ALARMS.PLC_PC_MAJOR_VERSIONS_MISMATCH_A := (("DB16005_U2_STA3_COAXIAL_CLIENT_INTERFACE".U2_STA3_CAM_Read.Variable."Version.Major" <> #VERSIONS_MAJOR) OR ("DB16000_OPC_UA_TRIGGER_ALARM".CLIENT.U2_STA3_COAXIAL.ALARMS.PLC_PC_MAJOR_VERSIONS_MISMATCH_A AND NOT "DB2120_MPP_ITC_IPC".RESET_FAULTS)) AND "DB7257_UNIT_2_STA_3_COAXIAL_ENABLE_DISABLE".ENABLED;
   "DB426_ALARMS_WARNINGS".ALARMS.UNIT_02.STATION_3_COAXIAL."720817" := "DB16000_OPC_UA_TRIGGER_ALARM".CLIENT.U2_STA3_COAXIAL.ALARMS.PLC_PC_MAJOR_VERSIONS_MISMATCH_A;
END_REGION

REGION Network 102: UNIT 2 STATION 3 COAXIAL CAMERA NO CAMERA AVAILABLE WARNING
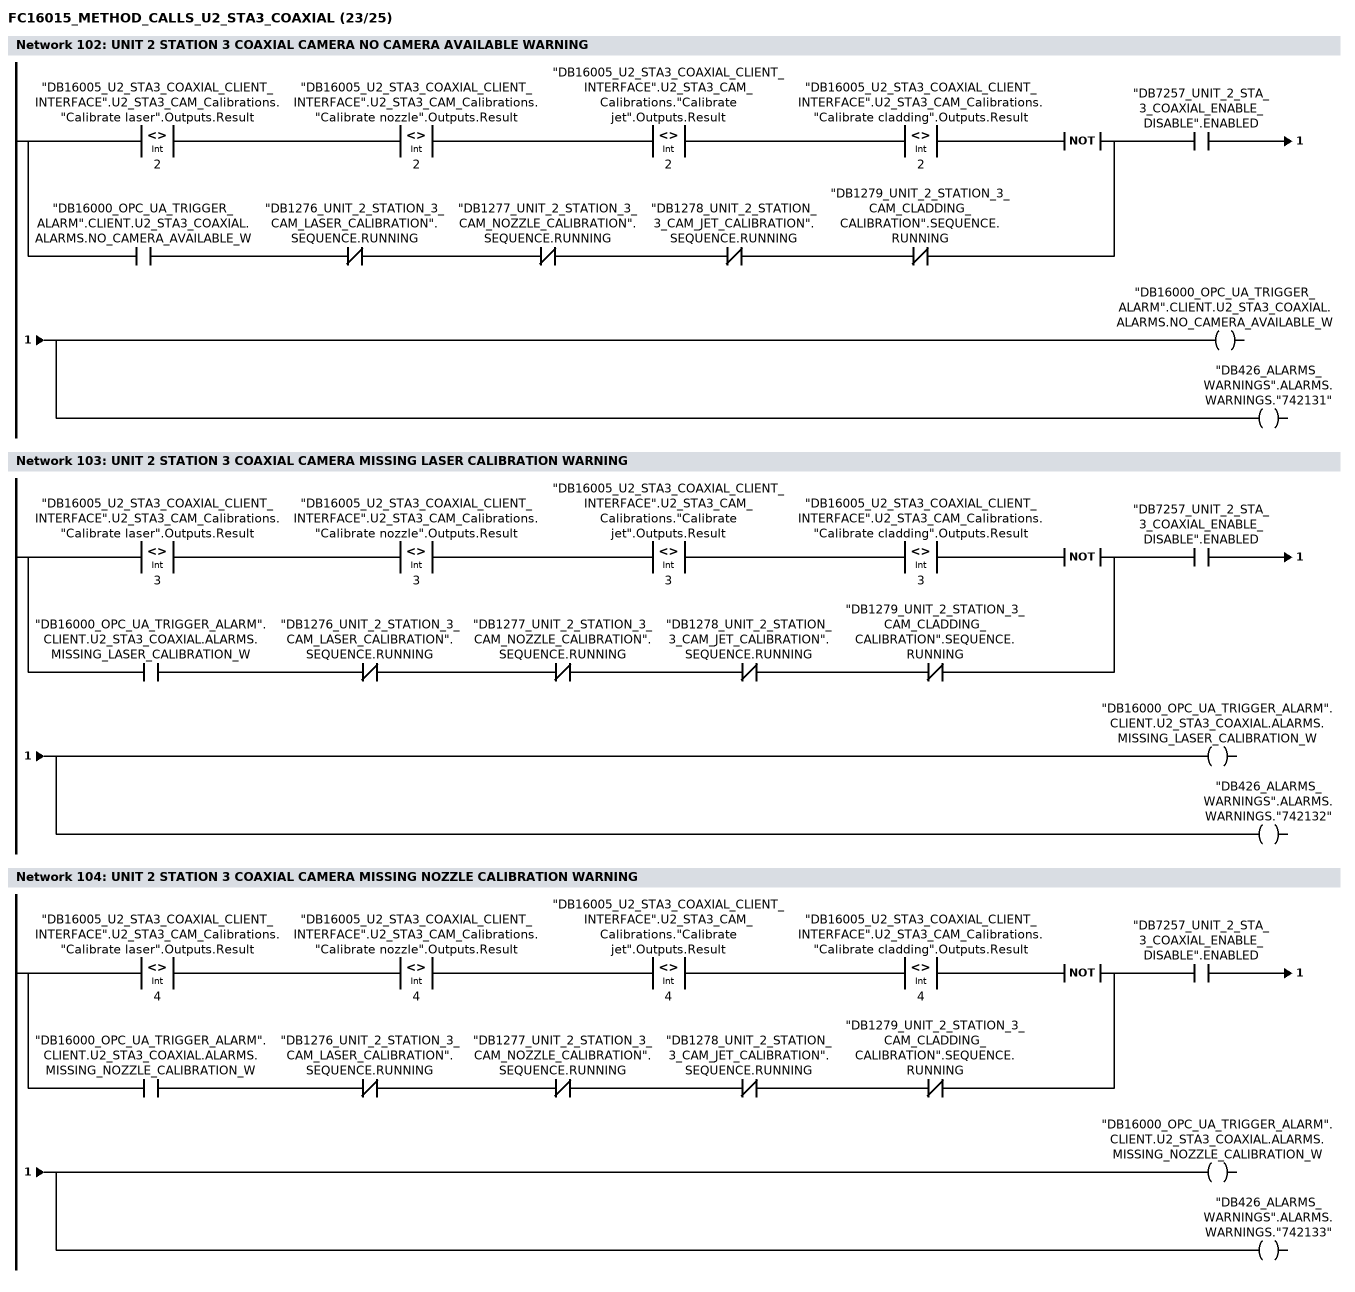
   RUNG wire#powerrail
      { S7_Templates := "SrcType := Int" } NE_Contact(in1 := "DB16005_U2_STA3_COAXIAL_CLIENT_INTERFACE".U2_STA3_CAM_Calibrations."Calibrate laser".Outputs.Result, in2 := 2)
      { S7_Templates := "SrcType := Int" } NE_Contact(in1 := "DB16005_U2_STA3_COAXIAL_CLIENT_INTERFACE".U2_STA3_CAM_Calibrations."Calibrate nozzle".Outputs.Result, in2 := 2)
      { S7_Templates := "SrcType := Int" } NE_Contact(in1 := "DB16005_U2_STA3_COAXIAL_CLIENT_INTERFACE".U2_STA3_CAM_Calibrations."Calibrate jet".Outputs.Result, in2 := 2)
      { S7_Templates := "SrcType := Int" } NE_Contact(in1 := "DB16005_U2_STA3_COAXIAL_CLIENT_INTERFACE".U2_STA3_CAM_Calibrations."Calibrate cladding".Outputs.Result, in2 := 2)
      Not()
      wire#w1
      Contact( "DB7257_UNIT_2_STA_3_COAXIAL_ENABLE_DISABLE".ENABLED )
      wire#w2
      Coil( "DB16000_OPC_UA_TRIGGER_ALARM".CLIENT.U2_STA3_COAXIAL.ALARMS.NO_CAMERA_AVAILABLE_W )
   END_RUNG
   RUNG wire#powerrail
      Contact( "DB16000_OPC_UA_TRIGGER_ALARM".CLIENT.U2_STA3_COAXIAL.ALARMS.NO_CAMERA_AVAILABLE_W )
      I_Contact( "DB1276_UNIT_2_STATION_3_CAM_LASER_CALIBRATION".SEQUENCE.RUNNING )
      I_Contact( "DB1277_UNIT_2_STATION_3_CAM_NOZZLE_CALIBRATION".SEQUENCE.RUNNING )
      I_Contact( "DB1278_UNIT_2_STATION_3_CAM_JET_CALIBRATION".SEQUENCE.RUNNING )
      I_Contact( "DB1279_UNIT_2_STATION_3_CAM_CLADDING_CALIBRATION".SEQUENCE.RUNNING )
   END_RUNG wire#w1
   RUNG wire#w2
      Coil( "DB426_ALARMS_WARNINGS".ALARMS.WARNINGS."742131" )
   END_RUNG
   // the same network as SCL:
   "DB16000_OPC_UA_TRIGGER_ALARM".CLIENT.U2_STA3_COAXIAL.ALARMS.NO_CAMERA_AVAILABLE_W := (NOT (("DB16005_U2_STA3_COAXIAL_CLIENT_INTERFACE".U2_STA3_CAM_Calibrations."Calibrate laser".Outputs.Result <> 2) AND ("DB16005_U2_STA3_COAXIAL_CLIENT_INTERFACE".U2_STA3_CAM_Calibrations."Calibrate nozzle".Outputs.Result <> 2) AND ("DB16005_U2_STA3_COAXIAL_CLIENT_INTERFACE".U2_STA3_CAM_Calibrations."Calibrate jet".Outputs.Result <> 2) AND ("DB16005_U2_STA3_COAXIAL_CLIENT_INTERFACE".U2_STA3_CAM_Calibrations."Calibrate cladding".Outputs.Result <> 2)) OR ("DB16000_OPC_UA_TRIGGER_ALARM".CLIENT.U2_STA3_COAXIAL.ALARMS.NO_CAMERA_AVAILABLE_W AND NOT "DB1276_UNIT_2_STATION_3_CAM_LASER_CALIBRATION".SEQUENCE.RUNNING AND NOT "DB1277_UNIT_2_STATION_3_CAM_NOZZLE_CALIBRATION".SEQUENCE.RUNNING AND NOT "DB1278_UNIT_2_STATION_3_CAM_JET_CALIBRATION".SEQUENCE.RUNNING AND NOT "DB1279_UNIT_2_STATION_3_CAM_CLADDING_CALIBRATION".SEQUENCE.RUNNING)) AND "DB7257_UNIT_2_STA_3_COAXIAL_ENABLE_DISABLE".ENABLED;
   "DB426_ALARMS_WARNINGS".ALARMS.WARNINGS."742131" := "DB16000_OPC_UA_TRIGGER_ALARM".CLIENT.U2_STA3_COAXIAL.ALARMS.NO_CAMERA_AVAILABLE_W;
END_REGION

REGION Network 103: UNIT 2 STATION 3 COAXIAL CAMERA MISSING LASER CALIBRATION WARNING
   RUNG wire#powerrail
      { S7_Templates := "SrcType := Int" } NE_Contact(in1 := "DB16005_U2_STA3_COAXIAL_CLIENT_INTERFACE".U2_STA3_CAM_Calibrations."Calibrate laser".Outputs.Result, in2 := 3)
      { S7_Templates := "SrcType := Int" } NE_Contact(in1 := "DB16005_U2_STA3_COAXIAL_CLIENT_INTERFACE".U2_STA3_CAM_Calibrations."Calibrate nozzle".Outputs.Result, in2 := 3)
      { S7_Templates := "SrcType := Int" } NE_Contact(in1 := "DB16005_U2_STA3_COAXIAL_CLIENT_INTERFACE".U2_STA3_CAM_Calibrations."Calibrate jet".Outputs.Result, in2 := 3)
      { S7_Templates := "SrcType := Int" } NE_Contact(in1 := "DB16005_U2_STA3_COAXIAL_CLIENT_INTERFACE".U2_STA3_CAM_Calibrations."Calibrate cladding".Outputs.Result, in2 := 3)
      Not()
      wire#w1
      Contact( "DB7257_UNIT_2_STA_3_COAXIAL_ENABLE_DISABLE".ENABLED )
      wire#w2
      Coil( "DB16000_OPC_UA_TRIGGER_ALARM".CLIENT.U2_STA3_COAXIAL.ALARMS.MISSING_LASER_CALIBRATION_W )
   END_RUNG
   RUNG wire#powerrail
      Contact( "DB16000_OPC_UA_TRIGGER_ALARM".CLIENT.U2_STA3_COAXIAL.ALARMS.MISSING_LASER_CALIBRATION_W )
      I_Contact( "DB1276_UNIT_2_STATION_3_CAM_LASER_CALIBRATION".SEQUENCE.RUNNING )
      I_Contact( "DB1277_UNIT_2_STATION_3_CAM_NOZZLE_CALIBRATION".SEQUENCE.RUNNING )
      I_Contact( "DB1278_UNIT_2_STATION_3_CAM_JET_CALIBRATION".SEQUENCE.RUNNING )
      I_Contact( "DB1279_UNIT_2_STATION_3_CAM_CLADDING_CALIBRATION".SEQUENCE.RUNNING )
   END_RUNG wire#w1
   RUNG wire#w2
      Coil( "DB426_ALARMS_WARNINGS".ALARMS.WARNINGS."742132" )
   END_RUNG
   // the same network as SCL:
   "DB16000_OPC_UA_TRIGGER_ALARM".CLIENT.U2_STA3_COAXIAL.ALARMS.MISSING_LASER_CALIBRATION_W := (NOT (("DB16005_U2_STA3_COAXIAL_CLIENT_INTERFACE".U2_STA3_CAM_Calibrations."Calibrate laser".Outputs.Result <> 3) AND ("DB16005_U2_STA3_COAXIAL_CLIENT_INTERFACE".U2_STA3_CAM_Calibrations."Calibrate nozzle".Outputs.Result <> 3) AND ("DB16005_U2_STA3_COAXIAL_CLIENT_INTERFACE".U2_STA3_CAM_Calibrations."Calibrate jet".Outputs.Result <> 3) AND ("DB16005_U2_STA3_COAXIAL_CLIENT_INTERFACE".U2_STA3_CAM_Calibrations."Calibrate cladding".Outputs.Result <> 3)) OR ("DB16000_OPC_UA_TRIGGER_ALARM".CLIENT.U2_STA3_COAXIAL.ALARMS.MISSING_LASER_CALIBRATION_W AND NOT "DB1276_UNIT_2_STATION_3_CAM_LASER_CALIBRATION".SEQUENCE.RUNNING AND NOT "DB1277_UNIT_2_STATION_3_CAM_NOZZLE_CALIBRATION".SEQUENCE.RUNNING AND NOT "DB1278_UNIT_2_STATION_3_CAM_JET_CALIBRATION".SEQUENCE.RUNNING AND NOT "DB1279_UNIT_2_STATION_3_CAM_CLADDING_CALIBRATION".SEQUENCE.RUNNING)) AND "DB7257_UNIT_2_STA_3_COAXIAL_ENABLE_DISABLE".ENABLED;
   "DB426_ALARMS_WARNINGS".ALARMS.WARNINGS."742132" := "DB16000_OPC_UA_TRIGGER_ALARM".CLIENT.U2_STA3_COAXIAL.ALARMS.MISSING_LASER_CALIBRATION_W;
END_REGION

REGION Network 104: UNIT 2 STATION 3 COAXIAL CAMERA MISSING NOZZLE CALIBRATION WARNING
   RUNG wire#powerrail
      { S7_Templates := "SrcType := Int" } NE_Contact(in1 := "DB16005_U2_STA3_COAXIAL_CLIENT_INTERFACE".U2_STA3_CAM_Calibrations."Calibrate laser".Outputs.Result, in2 := 4)
      { S7_Templates := "SrcType := Int" } NE_Contact(in1 := "DB16005_U2_STA3_COAXIAL_CLIENT_INTERFACE".U2_STA3_CAM_Calibrations."Calibrate nozzle".Outputs.Result, in2 := 4)
      { S7_Templates := "SrcType := Int" } NE_Contact(in1 := "DB16005_U2_STA3_COAXIAL_CLIENT_INTERFACE".U2_STA3_CAM_Calibrations."Calibrate jet".Outputs.Result, in2 := 4)
      { S7_Templates := "SrcType := Int" } NE_Contact(in1 := "DB16005_U2_STA3_COAXIAL_CLIENT_INTERFACE".U2_STA3_CAM_Calibrations."Calibrate cladding".Outputs.Result, in2 := 4)
      Not()
      wire#w1
      Contact( "DB7257_UNIT_2_STA_3_COAXIAL_ENABLE_DISABLE".ENABLED )
      wire#w2
      Coil( "DB16000_OPC_UA_TRIGGER_ALARM".CLIENT.U2_STA3_COAXIAL.ALARMS.MISSING_NOZZLE_CALIBRATION_W )
   END_RUNG
   RUNG wire#powerrail
      Contact( "DB16000_OPC_UA_TRIGGER_ALARM".CLIENT.U2_STA3_COAXIAL.ALARMS.MISSING_NOZZLE_CALIBRATION_W )
      I_Contact( "DB1276_UNIT_2_STATION_3_CAM_LASER_CALIBRATION".SEQUENCE.RUNNING )
      I_Contact( "DB1277_UNIT_2_STATION_3_CAM_NOZZLE_CALIBRATION".SEQUENCE.RUNNING )
      I_Contact( "DB1278_UNIT_2_STATION_3_CAM_JET_CALIBRATION".SEQUENCE.RUNNING )
      I_Contact( "DB1279_UNIT_2_STATION_3_CAM_CLADDING_CALIBRATION".SEQUENCE.RUNNING )
   END_RUNG wire#w1
   RUNG wire#w2
      Coil( "DB426_ALARMS_WARNINGS".ALARMS.WARNINGS."742133" )
   END_RUNG
   // the same network as SCL:
   "DB16000_OPC_UA_TRIGGER_ALARM".CLIENT.U2_STA3_COAXIAL.ALARMS.MISSING_NOZZLE_CALIBRATION_W := (NOT (("DB16005_U2_STA3_COAXIAL_CLIENT_INTERFACE".U2_STA3_CAM_Calibrations."Calibrate laser".Outputs.Result <> 4) AND ("DB16005_U2_STA3_COAXIAL_CLIENT_INTERFACE".U2_STA3_CAM_Calibrations."Calibrate nozzle".Outputs.Result <> 4) AND ("DB16005_U2_STA3_COAXIAL_CLIENT_INTERFACE".U2_STA3_CAM_Calibrations."Calibrate jet".Outputs.Result <> 4) AND ("DB16005_U2_STA3_COAXIAL_CLIENT_INTERFACE".U2_STA3_CAM_Calibrations."Calibrate cladding".Outputs.Result <> 4)) OR ("DB16000_OPC_UA_TRIGGER_ALARM".CLIENT.U2_STA3_COAXIAL.ALARMS.MISSING_NOZZLE_CALIBRATION_W AND NOT "DB1276_UNIT_2_STATION_3_CAM_LASER_CALIBRATION".SEQUENCE.RUNNING AND NOT "DB1277_UNIT_2_STATION_3_CAM_NOZZLE_CALIBRATION".SEQUENCE.RUNNING AND NOT "DB1278_UNIT_2_STATION_3_CAM_JET_CALIBRATION".SEQUENCE.RUNNING AND NOT "DB1279_UNIT_2_STATION_3_CAM_CLADDING_CALIBRATION".SEQUENCE.RUNNING)) AND "DB7257_UNIT_2_STA_3_COAXIAL_ENABLE_DISABLE".ENABLED;
   "DB426_ALARMS_WARNINGS".ALARMS.WARNINGS."742133" := "DB16000_OPC_UA_TRIGGER_ALARM".CLIENT.U2_STA3_COAXIAL.ALARMS.MISSING_NOZZLE_CALIBRATION_W;
END_REGION

REGION Network 105: IS_SEOC ALARMS
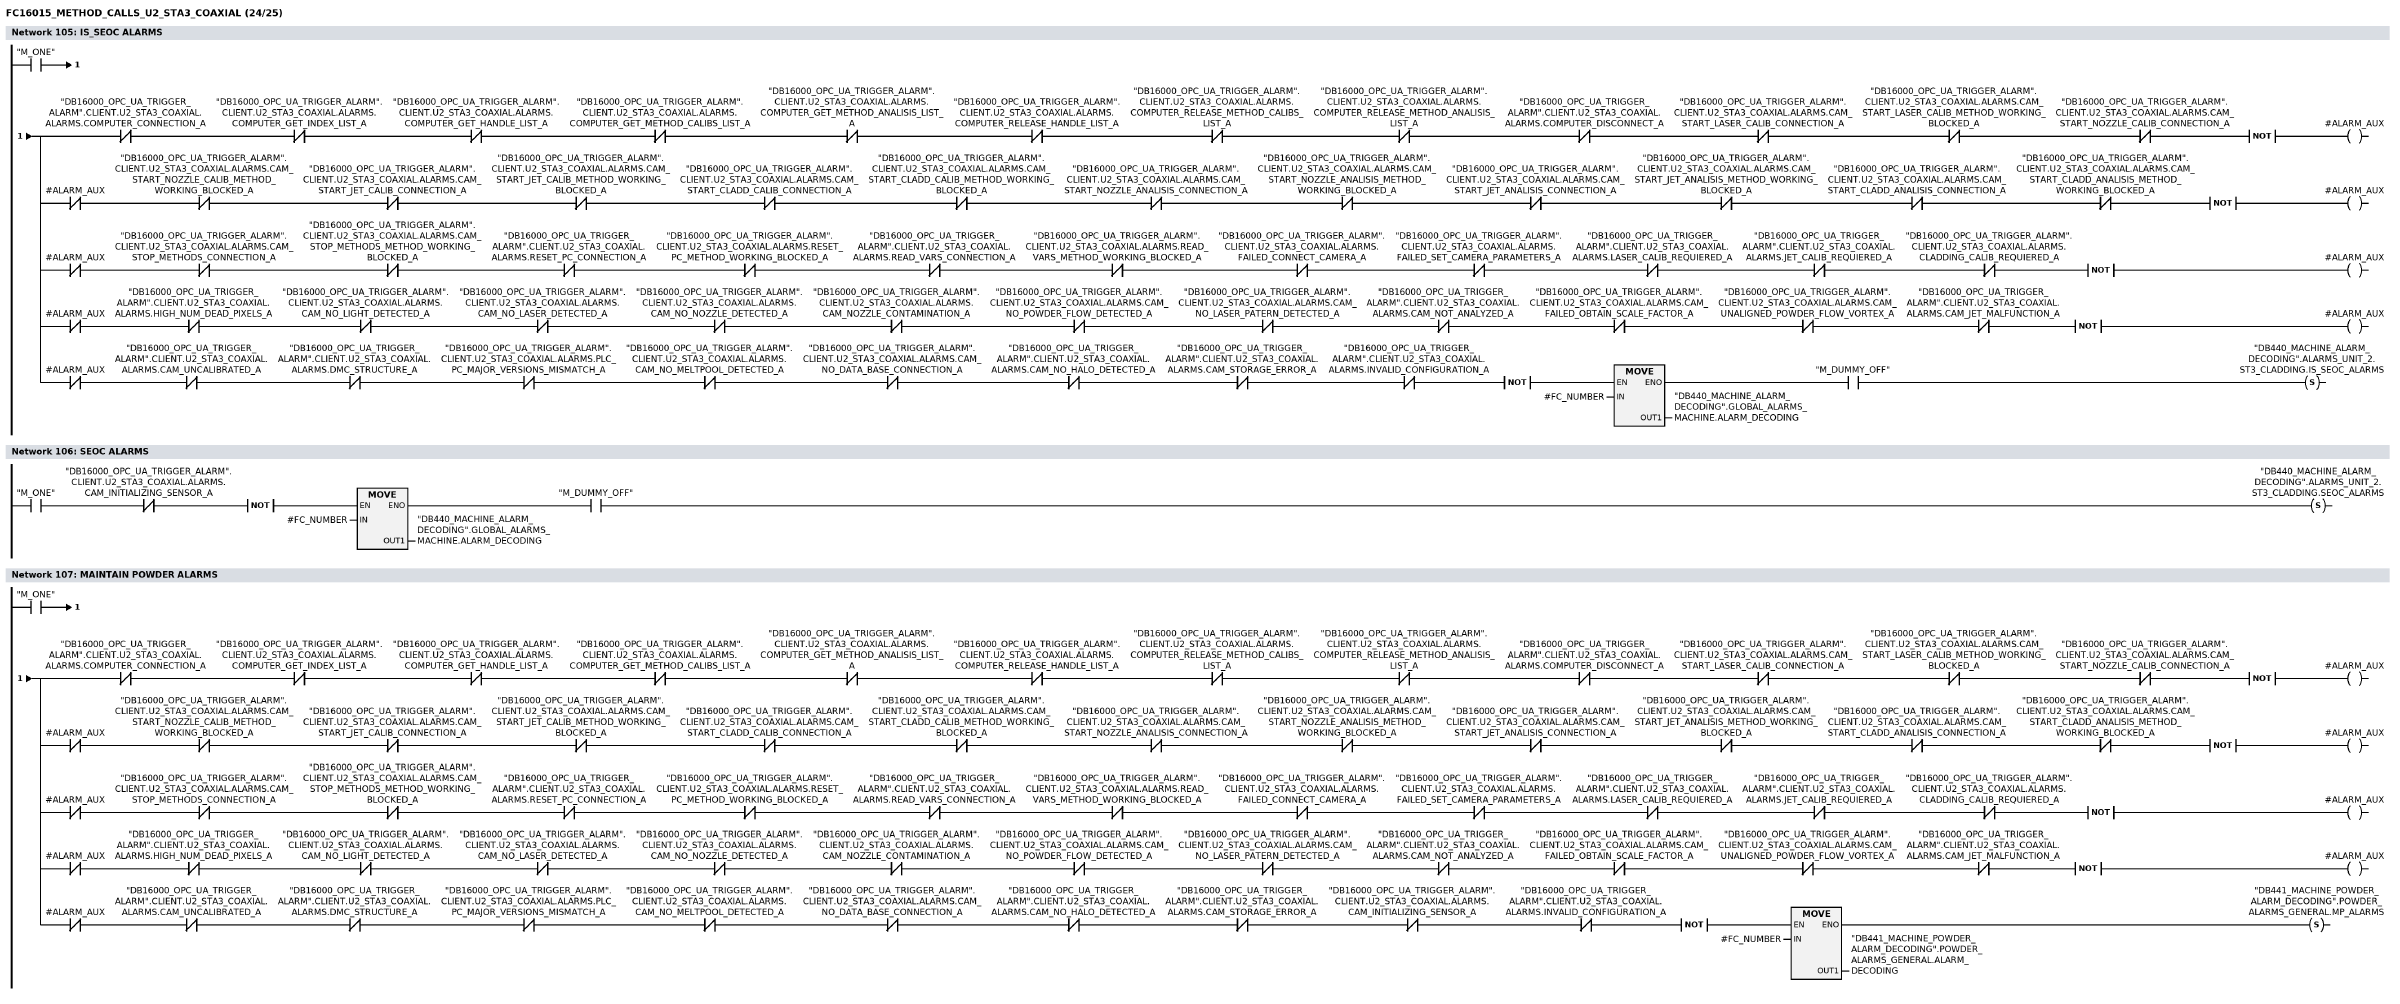
   RUNG wire#powerrail
      Contact( "M_ONE" )
      wire#w1
      I_Contact( "DB16000_OPC_UA_TRIGGER_ALARM".CLIENT.U2_STA3_COAXIAL.ALARMS.COMPUTER_CONNECTION_A )
      I_Contact( "DB16000_OPC_UA_TRIGGER_ALARM".CLIENT.U2_STA3_COAXIAL.ALARMS.COMPUTER_GET_INDEX_LIST_A )
      I_Contact( "DB16000_OPC_UA_TRIGGER_ALARM".CLIENT.U2_STA3_COAXIAL.ALARMS.COMPUTER_GET_HANDLE_LIST_A )
      I_Contact( "DB16000_OPC_UA_TRIGGER_ALARM".CLIENT.U2_STA3_COAXIAL.ALARMS.COMPUTER_GET_METHOD_CALIBS_LIST_A )
      I_Contact( "DB16000_OPC_UA_TRIGGER_ALARM".CLIENT.U2_STA3_COAXIAL.ALARMS.COMPUTER_GET_METHOD_ANALISIS_LIST_A )
      I_Contact( "DB16000_OPC_UA_TRIGGER_ALARM".CLIENT.U2_STA3_COAXIAL.ALARMS.COMPUTER_RELEASE_HANDLE_LIST_A )
      I_Contact( "DB16000_OPC_UA_TRIGGER_ALARM".CLIENT.U2_STA3_COAXIAL.ALARMS.COMPUTER_RELEASE_METHOD_CALIBS_LIST_A )
      I_Contact( "DB16000_OPC_UA_TRIGGER_ALARM".CLIENT.U2_STA3_COAXIAL.ALARMS.COMPUTER_RELEASE_METHOD_ANALISIS_LIST_A )
      I_Contact( "DB16000_OPC_UA_TRIGGER_ALARM".CLIENT.U2_STA3_COAXIAL.ALARMS.COMPUTER_DISCONNECT_A )
      I_Contact( "DB16000_OPC_UA_TRIGGER_ALARM".CLIENT.U2_STA3_COAXIAL.ALARMS.CAM_START_LASER_CALIB_CONNECTION_A )
      I_Contact( "DB16000_OPC_UA_TRIGGER_ALARM".CLIENT.U2_STA3_COAXIAL.ALARMS.CAM_START_LASER_CALIB_METHOD_WORKING_BLOCKED_A )
      I_Contact( "DB16000_OPC_UA_TRIGGER_ALARM".CLIENT.U2_STA3_COAXIAL.ALARMS.CAM_START_NOZZLE_CALIB_CONNECTION_A )
      Not()
      Coil( #ALARM_AUX )
   END_RUNG
   RUNG wire#w1
      I_Contact( #ALARM_AUX )
      I_Contact( "DB16000_OPC_UA_TRIGGER_ALARM".CLIENT.U2_STA3_COAXIAL.ALARMS.CAM_START_NOZZLE_CALIB_METHOD_WORKING_BLOCKED_A )
      I_Contact( "DB16000_OPC_UA_TRIGGER_ALARM".CLIENT.U2_STA3_COAXIAL.ALARMS.CAM_START_JET_CALIB_CONNECTION_A )
      I_Contact( "DB16000_OPC_UA_TRIGGER_ALARM".CLIENT.U2_STA3_COAXIAL.ALARMS.CAM_START_JET_CALIB_METHOD_WORKING_BLOCKED_A )
      I_Contact( "DB16000_OPC_UA_TRIGGER_ALARM".CLIENT.U2_STA3_COAXIAL.ALARMS.CAM_START_CLADD_CALIB_CONNECTION_A )
      I_Contact( "DB16000_OPC_UA_TRIGGER_ALARM".CLIENT.U2_STA3_COAXIAL.ALARMS.CAM_START_CLADD_CALIB_METHOD_WORKING_BLOCKED_A )
      I_Contact( "DB16000_OPC_UA_TRIGGER_ALARM".CLIENT.U2_STA3_COAXIAL.ALARMS.CAM_START_NOZZLE_ANALISIS_CONNECTION_A )
      I_Contact( "DB16000_OPC_UA_TRIGGER_ALARM".CLIENT.U2_STA3_COAXIAL.ALARMS.CAM_START_NOZZLE_ANALISIS_METHOD_WORKING_BLOCKED_A )
      I_Contact( "DB16000_OPC_UA_TRIGGER_ALARM".CLIENT.U2_STA3_COAXIAL.ALARMS.CAM_START_JET_ANALISIS_CONNECTION_A )
      I_Contact( "DB16000_OPC_UA_TRIGGER_ALARM".CLIENT.U2_STA3_COAXIAL.ALARMS.CAM_START_JET_ANALISIS_METHOD_WORKING_BLOCKED_A )
      I_Contact( "DB16000_OPC_UA_TRIGGER_ALARM".CLIENT.U2_STA3_COAXIAL.ALARMS.CAM_START_CLADD_ANALISIS_CONNECTION_A )
      I_Contact( "DB16000_OPC_UA_TRIGGER_ALARM".CLIENT.U2_STA3_COAXIAL.ALARMS.CAM_START_CLADD_ANALISIS_METHOD_WORKING_BLOCKED_A )
      Not()
      Coil( #ALARM_AUX )
   END_RUNG
   RUNG wire#w1
      I_Contact( #ALARM_AUX )
      I_Contact( "DB16000_OPC_UA_TRIGGER_ALARM".CLIENT.U2_STA3_COAXIAL.ALARMS.CAM_STOP_METHODS_CONNECTION_A )
      I_Contact( "DB16000_OPC_UA_TRIGGER_ALARM".CLIENT.U2_STA3_COAXIAL.ALARMS.CAM_STOP_METHODS_METHOD_WORKING_BLOCKED_A )
      I_Contact( "DB16000_OPC_UA_TRIGGER_ALARM".CLIENT.U2_STA3_COAXIAL.ALARMS.RESET_PC_CONNECTION_A )
      I_Contact( "DB16000_OPC_UA_TRIGGER_ALARM".CLIENT.U2_STA3_COAXIAL.ALARMS.RESET_PC_METHOD_WORKING_BLOCKED_A )
      I_Contact( "DB16000_OPC_UA_TRIGGER_ALARM".CLIENT.U2_STA3_COAXIAL.ALARMS.READ_VARS_CONNECTION_A )
      I_Contact( "DB16000_OPC_UA_TRIGGER_ALARM".CLIENT.U2_STA3_COAXIAL.ALARMS.READ_VARS_METHOD_WORKING_BLOCKED_A )
      I_Contact( "DB16000_OPC_UA_TRIGGER_ALARM".CLIENT.U2_STA3_COAXIAL.ALARMS.FAILED_CONNECT_CAMERA_A )
      I_Contact( "DB16000_OPC_UA_TRIGGER_ALARM".CLIENT.U2_STA3_COAXIAL.ALARMS.FAILED_SET_CAMERA_PARAMETERS_A )
      I_Contact( "DB16000_OPC_UA_TRIGGER_ALARM".CLIENT.U2_STA3_COAXIAL.ALARMS.LASER_CALIB_REQUIERED_A )
      I_Contact( "DB16000_OPC_UA_TRIGGER_ALARM".CLIENT.U2_STA3_COAXIAL.ALARMS.JET_CALIB_REQUIERED_A )
      I_Contact( "DB16000_OPC_UA_TRIGGER_ALARM".CLIENT.U2_STA3_COAXIAL.ALARMS.CLADDING_CALIB_REQUIERED_A )
      Not()
      Coil( #ALARM_AUX )
   END_RUNG
   RUNG wire#w1
      I_Contact( #ALARM_AUX )
      I_Contact( "DB16000_OPC_UA_TRIGGER_ALARM".CLIENT.U2_STA3_COAXIAL.ALARMS.HIGH_NUM_DEAD_PIXELS_A )
      I_Contact( "DB16000_OPC_UA_TRIGGER_ALARM".CLIENT.U2_STA3_COAXIAL.ALARMS.CAM_NO_LIGHT_DETECTED_A )
      I_Contact( "DB16000_OPC_UA_TRIGGER_ALARM".CLIENT.U2_STA3_COAXIAL.ALARMS.CAM_NO_LASER_DETECTED_A )
      I_Contact( "DB16000_OPC_UA_TRIGGER_ALARM".CLIENT.U2_STA3_COAXIAL.ALARMS.CAM_NO_NOZZLE_DETECTED_A )
      I_Contact( "DB16000_OPC_UA_TRIGGER_ALARM".CLIENT.U2_STA3_COAXIAL.ALARMS.CAM_NOZZLE_CONTAMINATION_A )
      I_Contact( "DB16000_OPC_UA_TRIGGER_ALARM".CLIENT.U2_STA3_COAXIAL.ALARMS.CAM_NO_POWDER_FLOW_DETECTED_A )
      I_Contact( "DB16000_OPC_UA_TRIGGER_ALARM".CLIENT.U2_STA3_COAXIAL.ALARMS.CAM_NO_LASER_PATERN_DETECTED_A )
      I_Contact( "DB16000_OPC_UA_TRIGGER_ALARM".CLIENT.U2_STA3_COAXIAL.ALARMS.CAM_NOT_ANALYZED_A )
      I_Contact( "DB16000_OPC_UA_TRIGGER_ALARM".CLIENT.U2_STA3_COAXIAL.ALARMS.CAM_FAILED_OBTAIN_SCALE_FACTOR_A )
      I_Contact( "DB16000_OPC_UA_TRIGGER_ALARM".CLIENT.U2_STA3_COAXIAL.ALARMS.CAM_UNALIGNED_POWDER_FLOW_VORTEX_A )
      I_Contact( "DB16000_OPC_UA_TRIGGER_ALARM".CLIENT.U2_STA3_COAXIAL.ALARMS.CAM_JET_MALFUNCTION_A )
      Not()
      Coil( #ALARM_AUX )
   END_RUNG
   RUNG wire#w1
      I_Contact( #ALARM_AUX )
      I_Contact( "DB16000_OPC_UA_TRIGGER_ALARM".CLIENT.U2_STA3_COAXIAL.ALARMS.CAM_UNCALIBRATED_A )
      I_Contact( "DB16000_OPC_UA_TRIGGER_ALARM".CLIENT.U2_STA3_COAXIAL.ALARMS.DMC_STRUCTURE_A )
      I_Contact( "DB16000_OPC_UA_TRIGGER_ALARM".CLIENT.U2_STA3_COAXIAL.ALARMS.PLC_PC_MAJOR_VERSIONS_MISMATCH_A )
      I_Contact( "DB16000_OPC_UA_TRIGGER_ALARM".CLIENT.U2_STA3_COAXIAL.ALARMS.CAM_NO_MELTPOOL_DETECTED_A )
      I_Contact( "DB16000_OPC_UA_TRIGGER_ALARM".CLIENT.U2_STA3_COAXIAL.ALARMS.CAM_NO_DATA_BASE_CONNECTION_A )
      I_Contact( "DB16000_OPC_UA_TRIGGER_ALARM".CLIENT.U2_STA3_COAXIAL.ALARMS.CAM_NO_HALO_DETECTED_A )
      I_Contact( "DB16000_OPC_UA_TRIGGER_ALARM".CLIENT.U2_STA3_COAXIAL.ALARMS.CAM_STORAGE_ERROR_A )
      I_Contact( "DB16000_OPC_UA_TRIGGER_ALARM".CLIENT.U2_STA3_COAXIAL.ALARMS.INVALID_CONFIGURATION_A )
      Not()
      Move(in := #FC_NUMBER, out1 => "DB440_MACHINE_ALARM_DECODING".GLOBAL_ALARMS_MACHINE.ALARM_DECODING)
      Contact( "M_DUMMY_OFF" )
      S_Coil( "DB440_MACHINE_ALARM_DECODING".ALARMS_UNIT_2.ST3_CLADDING.IS_SEOC_ALARMS )
   END_RUNG
   // the same network as SCL:
   #ALARM_AUX := NOT ("M_ONE" AND NOT "DB16000_OPC_UA_TRIGGER_ALARM".CLIENT.U2_STA3_COAXIAL.ALARMS.COMPUTER_CONNECTION_A AND NOT "DB16000_OPC_UA_TRIGGER_ALARM".CLIENT.U2_STA3_COAXIAL.ALARMS.COMPUTER_GET_INDEX_LIST_A AND NOT "DB16000_OPC_UA_TRIGGER_ALARM".CLIENT.U2_STA3_COAXIAL.ALARMS.COMPUTER_GET_HANDLE_LIST_A AND NOT "DB16000_OPC_UA_TRIGGER_ALARM".CLIENT.U2_STA3_COAXIAL.ALARMS.COMPUTER_GET_METHOD_CALIBS_LIST_A AND NOT "DB16000_OPC_UA_TRIGGER_ALARM".CLIENT.U2_STA3_COAXIAL.ALARMS.COMPUTER_GET_METHOD_ANALISIS_LIST_A AND NOT "DB16000_OPC_UA_TRIGGER_ALARM".CLIENT.U2_STA3_COAXIAL.ALARMS.COMPUTER_RELEASE_HANDLE_LIST_A AND NOT "DB16000_OPC_UA_TRIGGER_ALARM".CLIENT.U2_STA3_COAXIAL.ALARMS.COMPUTER_RELEASE_METHOD_CALIBS_LIST_A AND NOT "DB16000_OPC_UA_TRIGGER_ALARM".CLIENT.U2_STA3_COAXIAL.ALARMS.COMPUTER_RELEASE_METHOD_ANALISIS_LIST_A AND NOT "DB16000_OPC_UA_TRIGGER_ALARM".CLIENT.U2_STA3_COAXIAL.ALARMS.COMPUTER_DISCONNECT_A AND NOT "DB16000_OPC_UA_TRIGGER_ALARM".CLIENT.U2_STA3_COAXIAL.ALARMS.CAM_START_LASER_CALIB_CONNECTION_A AND NOT "DB16000_OPC_UA_TRIGGER_ALARM".CLIENT.U2_STA3_COAXIAL.ALARMS.CAM_START_LASER_CALIB_METHOD_WORKING_BLOCKED_A AND NOT "DB16000_OPC_UA_TRIGGER_ALARM".CLIENT.U2_STA3_COAXIAL.ALARMS.CAM_START_NOZZLE_CALIB_CONNECTION_A);
   #ALARM_AUX := NOT ("M_ONE" AND NOT #ALARM_AUX AND NOT "DB16000_OPC_UA_TRIGGER_ALARM".CLIENT.U2_STA3_COAXIAL.ALARMS.CAM_START_NOZZLE_CALIB_METHOD_WORKING_BLOCKED_A AND NOT "DB16000_OPC_UA_TRIGGER_ALARM".CLIENT.U2_STA3_COAXIAL.ALARMS.CAM_START_JET_CALIB_CONNECTION_A AND NOT "DB16000_OPC_UA_TRIGGER_ALARM".CLIENT.U2_STA3_COAXIAL.ALARMS.CAM_START_JET_CALIB_METHOD_WORKING_BLOCKED_A AND NOT "DB16000_OPC_UA_TRIGGER_ALARM".CLIENT.U2_STA3_COAXIAL.ALARMS.CAM_START_CLADD_CALIB_CONNECTION_A AND NOT "DB16000_OPC_UA_TRIGGER_ALARM".CLIENT.U2_STA3_COAXIAL.ALARMS.CAM_START_CLADD_CALIB_METHOD_WORKING_BLOCKED_A AND NOT "DB16000_OPC_UA_TRIGGER_ALARM".CLIENT.U2_STA3_COAXIAL.ALARMS.CAM_START_NOZZLE_ANALISIS_CONNECTION_A AND NOT "DB16000_OPC_UA_TRIGGER_ALARM".CLIENT.U2_STA3_COAXIAL.ALARMS.CAM_START_NOZZLE_ANALISIS_METHOD_WORKING_BLOCKED_A AND NOT "DB16000_OPC_UA_TRIGGER_ALARM".CLIENT.U2_STA3_COAXIAL.ALARMS.CAM_START_JET_ANALISIS_CONNECTION_A AND NOT "DB16000_OPC_UA_TRIGGER_ALARM".CLIENT.U2_STA3_COAXIAL.ALARMS.CAM_START_JET_ANALISIS_METHOD_WORKING_BLOCKED_A AND NOT "DB16000_OPC_UA_TRIGGER_ALARM".CLIENT.U2_STA3_COAXIAL.ALARMS.CAM_START_CLADD_ANALISIS_CONNECTION_A AND NOT "DB16000_OPC_UA_TRIGGER_ALARM".CLIENT.U2_STA3_COAXIAL.ALARMS.CAM_START_CLADD_ANALISIS_METHOD_WORKING_BLOCKED_A);
   #ALARM_AUX := NOT ("M_ONE" AND NOT #ALARM_AUX AND NOT "DB16000_OPC_UA_TRIGGER_ALARM".CLIENT.U2_STA3_COAXIAL.ALARMS.CAM_STOP_METHODS_CONNECTION_A AND NOT "DB16000_OPC_UA_TRIGGER_ALARM".CLIENT.U2_STA3_COAXIAL.ALARMS.CAM_STOP_METHODS_METHOD_WORKING_BLOCKED_A AND NOT "DB16000_OPC_UA_TRIGGER_ALARM".CLIENT.U2_STA3_COAXIAL.ALARMS.RESET_PC_CONNECTION_A AND NOT "DB16000_OPC_UA_TRIGGER_ALARM".CLIENT.U2_STA3_COAXIAL.ALARMS.RESET_PC_METHOD_WORKING_BLOCKED_A AND NOT "DB16000_OPC_UA_TRIGGER_ALARM".CLIENT.U2_STA3_COAXIAL.ALARMS.READ_VARS_CONNECTION_A AND NOT "DB16000_OPC_UA_TRIGGER_ALARM".CLIENT.U2_STA3_COAXIAL.ALARMS.READ_VARS_METHOD_WORKING_BLOCKED_A AND NOT "DB16000_OPC_UA_TRIGGER_ALARM".CLIENT.U2_STA3_COAXIAL.ALARMS.FAILED_CONNECT_CAMERA_A AND NOT "DB16000_OPC_UA_TRIGGER_ALARM".CLIENT.U2_STA3_COAXIAL.ALARMS.FAILED_SET_CAMERA_PARAMETERS_A AND NOT "DB16000_OPC_UA_TRIGGER_ALARM".CLIENT.U2_STA3_COAXIAL.ALARMS.LASER_CALIB_REQUIERED_A AND NOT "DB16000_OPC_UA_TRIGGER_ALARM".CLIENT.U2_STA3_COAXIAL.ALARMS.JET_CALIB_REQUIERED_A AND NOT "DB16000_OPC_UA_TRIGGER_ALARM".CLIENT.U2_STA3_COAXIAL.ALARMS.CLADDING_CALIB_REQUIERED_A);
   #ALARM_AUX := NOT ("M_ONE" AND NOT #ALARM_AUX AND NOT "DB16000_OPC_UA_TRIGGER_ALARM".CLIENT.U2_STA3_COAXIAL.ALARMS.HIGH_NUM_DEAD_PIXELS_A AND NOT "DB16000_OPC_UA_TRIGGER_ALARM".CLIENT.U2_STA3_COAXIAL.ALARMS.CAM_NO_LIGHT_DETECTED_A AND NOT "DB16000_OPC_UA_TRIGGER_ALARM".CLIENT.U2_STA3_COAXIAL.ALARMS.CAM_NO_LASER_DETECTED_A AND NOT "DB16000_OPC_UA_TRIGGER_ALARM".CLIENT.U2_STA3_COAXIAL.ALARMS.CAM_NO_NOZZLE_DETECTED_A AND NOT "DB16000_OPC_UA_TRIGGER_ALARM".CLIENT.U2_STA3_COAXIAL.ALARMS.CAM_NOZZLE_CONTAMINATION_A AND NOT "DB16000_OPC_UA_TRIGGER_ALARM".CLIENT.U2_STA3_COAXIAL.ALARMS.CAM_NO_POWDER_FLOW_DETECTED_A AND NOT "DB16000_OPC_UA_TRIGGER_ALARM".CLIENT.U2_STA3_COAXIAL.ALARMS.CAM_NO_LASER_PATERN_DETECTED_A AND NOT "DB16000_OPC_UA_TRIGGER_ALARM".CLIENT.U2_STA3_COAXIAL.ALARMS.CAM_NOT_ANALYZED_A AND NOT "DB16000_OPC_UA_TRIGGER_ALARM".CLIENT.U2_STA3_COAXIAL.ALARMS.CAM_FAILED_OBTAIN_SCALE_FACTOR_A AND NOT "DB16000_OPC_UA_TRIGGER_ALARM".CLIENT.U2_STA3_COAXIAL.ALARMS.CAM_UNALIGNED_POWDER_FLOW_VORTEX_A AND NOT "DB16000_OPC_UA_TRIGGER_ALARM".CLIENT.U2_STA3_COAXIAL.ALARMS.CAM_JET_MALFUNCTION_A);
   #_w1 := NOT ("M_ONE" AND NOT #ALARM_AUX AND NOT "DB16000_OPC_UA_TRIGGER_ALARM".CLIENT.U2_STA3_COAXIAL.ALARMS.CAM_UNCALIBRATED_A AND NOT "DB16000_OPC_UA_TRIGGER_ALARM".CLIENT.U2_STA3_COAXIAL.ALARMS.DMC_STRUCTURE_A AND NOT "DB16000_OPC_UA_TRIGGER_ALARM".CLIENT.U2_STA3_COAXIAL.ALARMS.PLC_PC_MAJOR_VERSIONS_MISMATCH_A AND NOT "DB16000_OPC_UA_TRIGGER_ALARM".CLIENT.U2_STA3_COAXIAL.ALARMS.CAM_NO_MELTPOOL_DETECTED_A AND NOT "DB16000_OPC_UA_TRIGGER_ALARM".CLIENT.U2_STA3_COAXIAL.ALARMS.CAM_NO_DATA_BASE_CONNECTION_A AND NOT "DB16000_OPC_UA_TRIGGER_ALARM".CLIENT.U2_STA3_COAXIAL.ALARMS.CAM_NO_HALO_DETECTED_A AND NOT "DB16000_OPC_UA_TRIGGER_ALARM".CLIENT.U2_STA3_COAXIAL.ALARMS.CAM_STORAGE_ERROR_A AND NOT "DB16000_OPC_UA_TRIGGER_ALARM".CLIENT.U2_STA3_COAXIAL.ALARMS.INVALID_CONFIGURATION_A);
   IF #_w1 THEN "DB440_MACHINE_ALARM_DECODING".GLOBAL_ALARMS_MACHINE.ALARM_DECODING := #FC_NUMBER; END_IF;
   IF #_w1 AND "M_DUMMY_OFF" THEN
       "DB440_MACHINE_ALARM_DECODING".ALARMS_UNIT_2.ST3_CLADDING.IS_SEOC_ALARMS := TRUE;
   END_IF;
END_REGION

REGION Network 106: SEOC ALARMS
   RUNG wire#powerrail
      Contact( "M_ONE" )
      I_Contact( "DB16000_OPC_UA_TRIGGER_ALARM".CLIENT.U2_STA3_COAXIAL.ALARMS.CAM_INITIALIZING_SENSOR_A )
      Not()
      Move(in := #FC_NUMBER, out1 => "DB440_MACHINE_ALARM_DECODING".GLOBAL_ALARMS_MACHINE.ALARM_DECODING)
      Contact( "M_DUMMY_OFF" )
      S_Coil( "DB440_MACHINE_ALARM_DECODING".ALARMS_UNIT_2.ST3_CLADDING.SEOC_ALARMS )
   END_RUNG
   // the same network as SCL:
   #_w1 := NOT ("M_ONE" AND NOT "DB16000_OPC_UA_TRIGGER_ALARM".CLIENT.U2_STA3_COAXIAL.ALARMS.CAM_INITIALIZING_SENSOR_A);
   IF #_w1 THEN "DB440_MACHINE_ALARM_DECODING".GLOBAL_ALARMS_MACHINE.ALARM_DECODING := #FC_NUMBER; END_IF;
   IF #_w1 AND "M_DUMMY_OFF" THEN
       "DB440_MACHINE_ALARM_DECODING".ALARMS_UNIT_2.ST3_CLADDING.SEOC_ALARMS := TRUE;
   END_IF;
END_REGION

REGION Network 107: MAINTAIN POWDER ALARMS
   RUNG wire#powerrail
      Contact( "M_ONE" )
      wire#w1
      I_Contact( "DB16000_OPC_UA_TRIGGER_ALARM".CLIENT.U2_STA3_COAXIAL.ALARMS.COMPUTER_CONNECTION_A )
      I_Contact( "DB16000_OPC_UA_TRIGGER_ALARM".CLIENT.U2_STA3_COAXIAL.ALARMS.COMPUTER_GET_INDEX_LIST_A )
      I_Contact( "DB16000_OPC_UA_TRIGGER_ALARM".CLIENT.U2_STA3_COAXIAL.ALARMS.COMPUTER_GET_HANDLE_LIST_A )
      I_Contact( "DB16000_OPC_UA_TRIGGER_ALARM".CLIENT.U2_STA3_COAXIAL.ALARMS.COMPUTER_GET_METHOD_CALIBS_LIST_A )
      I_Contact( "DB16000_OPC_UA_TRIGGER_ALARM".CLIENT.U2_STA3_COAXIAL.ALARMS.COMPUTER_GET_METHOD_ANALISIS_LIST_A )
      I_Contact( "DB16000_OPC_UA_TRIGGER_ALARM".CLIENT.U2_STA3_COAXIAL.ALARMS.COMPUTER_RELEASE_HANDLE_LIST_A )
      I_Contact( "DB16000_OPC_UA_TRIGGER_ALARM".CLIENT.U2_STA3_COAXIAL.ALARMS.COMPUTER_RELEASE_METHOD_CALIBS_LIST_A )
      I_Contact( "DB16000_OPC_UA_TRIGGER_ALARM".CLIENT.U2_STA3_COAXIAL.ALARMS.COMPUTER_RELEASE_METHOD_ANALISIS_LIST_A )
      I_Contact( "DB16000_OPC_UA_TRIGGER_ALARM".CLIENT.U2_STA3_COAXIAL.ALARMS.COMPUTER_DISCONNECT_A )
      I_Contact( "DB16000_OPC_UA_TRIGGER_ALARM".CLIENT.U2_STA3_COAXIAL.ALARMS.CAM_START_LASER_CALIB_CONNECTION_A )
      I_Contact( "DB16000_OPC_UA_TRIGGER_ALARM".CLIENT.U2_STA3_COAXIAL.ALARMS.CAM_START_LASER_CALIB_METHOD_WORKING_BLOCKED_A )
      I_Contact( "DB16000_OPC_UA_TRIGGER_ALARM".CLIENT.U2_STA3_COAXIAL.ALARMS.CAM_START_NOZZLE_CALIB_CONNECTION_A )
      Not()
      Coil( #ALARM_AUX )
   END_RUNG
   RUNG wire#w1
      I_Contact( #ALARM_AUX )
      I_Contact( "DB16000_OPC_UA_TRIGGER_ALARM".CLIENT.U2_STA3_COAXIAL.ALARMS.CAM_START_NOZZLE_CALIB_METHOD_WORKING_BLOCKED_A )
      I_Contact( "DB16000_OPC_UA_TRIGGER_ALARM".CLIENT.U2_STA3_COAXIAL.ALARMS.CAM_START_JET_CALIB_CONNECTION_A )
      I_Contact( "DB16000_OPC_UA_TRIGGER_ALARM".CLIENT.U2_STA3_COAXIAL.ALARMS.CAM_START_JET_CALIB_METHOD_WORKING_BLOCKED_A )
      I_Contact( "DB16000_OPC_UA_TRIGGER_ALARM".CLIENT.U2_STA3_COAXIAL.ALARMS.CAM_START_CLADD_CALIB_CONNECTION_A )
      I_Contact( "DB16000_OPC_UA_TRIGGER_ALARM".CLIENT.U2_STA3_COAXIAL.ALARMS.CAM_START_CLADD_CALIB_METHOD_WORKING_BLOCKED_A )
      I_Contact( "DB16000_OPC_UA_TRIGGER_ALARM".CLIENT.U2_STA3_COAXIAL.ALARMS.CAM_START_NOZZLE_ANALISIS_CONNECTION_A )
      I_Contact( "DB16000_OPC_UA_TRIGGER_ALARM".CLIENT.U2_STA3_COAXIAL.ALARMS.CAM_START_NOZZLE_ANALISIS_METHOD_WORKING_BLOCKED_A )
      I_Contact( "DB16000_OPC_UA_TRIGGER_ALARM".CLIENT.U2_STA3_COAXIAL.ALARMS.CAM_START_JET_ANALISIS_CONNECTION_A )
      I_Contact( "DB16000_OPC_UA_TRIGGER_ALARM".CLIENT.U2_STA3_COAXIAL.ALARMS.CAM_START_JET_ANALISIS_METHOD_WORKING_BLOCKED_A )
      I_Contact( "DB16000_OPC_UA_TRIGGER_ALARM".CLIENT.U2_STA3_COAXIAL.ALARMS.CAM_START_CLADD_ANALISIS_CONNECTION_A )
      I_Contact( "DB16000_OPC_UA_TRIGGER_ALARM".CLIENT.U2_STA3_COAXIAL.ALARMS.CAM_START_CLADD_ANALISIS_METHOD_WORKING_BLOCKED_A )
      Not()
      Coil( #ALARM_AUX )
   END_RUNG
   RUNG wire#w1
      I_Contact( #ALARM_AUX )
      I_Contact( "DB16000_OPC_UA_TRIGGER_ALARM".CLIENT.U2_STA3_COAXIAL.ALARMS.CAM_STOP_METHODS_CONNECTION_A )
      I_Contact( "DB16000_OPC_UA_TRIGGER_ALARM".CLIENT.U2_STA3_COAXIAL.ALARMS.CAM_STOP_METHODS_METHOD_WORKING_BLOCKED_A )
      I_Contact( "DB16000_OPC_UA_TRIGGER_ALARM".CLIENT.U2_STA3_COAXIAL.ALARMS.RESET_PC_CONNECTION_A )
      I_Contact( "DB16000_OPC_UA_TRIGGER_ALARM".CLIENT.U2_STA3_COAXIAL.ALARMS.RESET_PC_METHOD_WORKING_BLOCKED_A )
      I_Contact( "DB16000_OPC_UA_TRIGGER_ALARM".CLIENT.U2_STA3_COAXIAL.ALARMS.READ_VARS_CONNECTION_A )
      I_Contact( "DB16000_OPC_UA_TRIGGER_ALARM".CLIENT.U2_STA3_COAXIAL.ALARMS.READ_VARS_METHOD_WORKING_BLOCKED_A )
      I_Contact( "DB16000_OPC_UA_TRIGGER_ALARM".CLIENT.U2_STA3_COAXIAL.ALARMS.FAILED_CONNECT_CAMERA_A )
      I_Contact( "DB16000_OPC_UA_TRIGGER_ALARM".CLIENT.U2_STA3_COAXIAL.ALARMS.FAILED_SET_CAMERA_PARAMETERS_A )
      I_Contact( "DB16000_OPC_UA_TRIGGER_ALARM".CLIENT.U2_STA3_COAXIAL.ALARMS.LASER_CALIB_REQUIERED_A )
      I_Contact( "DB16000_OPC_UA_TRIGGER_ALARM".CLIENT.U2_STA3_COAXIAL.ALARMS.JET_CALIB_REQUIERED_A )
      I_Contact( "DB16000_OPC_UA_TRIGGER_ALARM".CLIENT.U2_STA3_COAXIAL.ALARMS.CLADDING_CALIB_REQUIERED_A )
      Not()
      Coil( #ALARM_AUX )
   END_RUNG
   RUNG wire#w1
      I_Contact( #ALARM_AUX )
      I_Contact( "DB16000_OPC_UA_TRIGGER_ALARM".CLIENT.U2_STA3_COAXIAL.ALARMS.HIGH_NUM_DEAD_PIXELS_A )
      I_Contact( "DB16000_OPC_UA_TRIGGER_ALARM".CLIENT.U2_STA3_COAXIAL.ALARMS.CAM_NO_LIGHT_DETECTED_A )
      I_Contact( "DB16000_OPC_UA_TRIGGER_ALARM".CLIENT.U2_STA3_COAXIAL.ALARMS.CAM_NO_LASER_DETECTED_A )
      I_Contact( "DB16000_OPC_UA_TRIGGER_ALARM".CLIENT.U2_STA3_COAXIAL.ALARMS.CAM_NO_NOZZLE_DETECTED_A )
      I_Contact( "DB16000_OPC_UA_TRIGGER_ALARM".CLIENT.U2_STA3_COAXIAL.ALARMS.CAM_NOZZLE_CONTAMINATION_A )
      I_Contact( "DB16000_OPC_UA_TRIGGER_ALARM".CLIENT.U2_STA3_COAXIAL.ALARMS.CAM_NO_POWDER_FLOW_DETECTED_A )
      I_Contact( "DB16000_OPC_UA_TRIGGER_ALARM".CLIENT.U2_STA3_COAXIAL.ALARMS.CAM_NO_LASER_PATERN_DETECTED_A )
      I_Contact( "DB16000_OPC_UA_TRIGGER_ALARM".CLIENT.U2_STA3_COAXIAL.ALARMS.CAM_NOT_ANALYZED_A )
      I_Contact( "DB16000_OPC_UA_TRIGGER_ALARM".CLIENT.U2_STA3_COAXIAL.ALARMS.CAM_FAILED_OBTAIN_SCALE_FACTOR_A )
      I_Contact( "DB16000_OPC_UA_TRIGGER_ALARM".CLIENT.U2_STA3_COAXIAL.ALARMS.CAM_UNALIGNED_POWDER_FLOW_VORTEX_A )
      I_Contact( "DB16000_OPC_UA_TRIGGER_ALARM".CLIENT.U2_STA3_COAXIAL.ALARMS.CAM_JET_MALFUNCTION_A )
      Not()
      Coil( #ALARM_AUX )
   END_RUNG
   RUNG wire#w1
      I_Contact( #ALARM_AUX )
      I_Contact( "DB16000_OPC_UA_TRIGGER_ALARM".CLIENT.U2_STA3_COAXIAL.ALARMS.CAM_UNCALIBRATED_A )
      I_Contact( "DB16000_OPC_UA_TRIGGER_ALARM".CLIENT.U2_STA3_COAXIAL.ALARMS.DMC_STRUCTURE_A )
      I_Contact( "DB16000_OPC_UA_TRIGGER_ALARM".CLIENT.U2_STA3_COAXIAL.ALARMS.PLC_PC_MAJOR_VERSIONS_MISMATCH_A )
      I_Contact( "DB16000_OPC_UA_TRIGGER_ALARM".CLIENT.U2_STA3_COAXIAL.ALARMS.CAM_NO_MELTPOOL_DETECTED_A )
      I_Contact( "DB16000_OPC_UA_TRIGGER_ALARM".CLIENT.U2_STA3_COAXIAL.ALARMS.CAM_NO_DATA_BASE_CONNECTION_A )
      I_Contact( "DB16000_OPC_UA_TRIGGER_ALARM".CLIENT.U2_STA3_COAXIAL.ALARMS.CAM_NO_HALO_DETECTED_A )
      I_Contact( "DB16000_OPC_UA_TRIGGER_ALARM".CLIENT.U2_STA3_COAXIAL.ALARMS.CAM_STORAGE_ERROR_A )
      I_Contact( "DB16000_OPC_UA_TRIGGER_ALARM".CLIENT.U2_STA3_COAXIAL.ALARMS.CAM_INITIALIZING_SENSOR_A )
      I_Contact( "DB16000_OPC_UA_TRIGGER_ALARM".CLIENT.U2_STA3_COAXIAL.ALARMS.INVALID_CONFIGURATION_A )
      Not()
      Move(in := #FC_NUMBER, out1 => "DB441_MACHINE_POWDER_ALARM_DECODING".POWDER_ALARMS_GENERAL.ALARM_DECODING)
      S_Coil( "DB441_MACHINE_POWDER_ALARM_DECODING".POWDER_ALARMS_GENERAL.MP_ALARMS )
   END_RUNG
   // the same network as SCL:
   #ALARM_AUX := NOT ("M_ONE" AND NOT "DB16000_OPC_UA_TRIGGER_ALARM".CLIENT.U2_STA3_COAXIAL.ALARMS.COMPUTER_CONNECTION_A AND NOT "DB16000_OPC_UA_TRIGGER_ALARM".CLIENT.U2_STA3_COAXIAL.ALARMS.COMPUTER_GET_INDEX_LIST_A AND NOT "DB16000_OPC_UA_TRIGGER_ALARM".CLIENT.U2_STA3_COAXIAL.ALARMS.COMPUTER_GET_HANDLE_LIST_A AND NOT "DB16000_OPC_UA_TRIGGER_ALARM".CLIENT.U2_STA3_COAXIAL.ALARMS.COMPUTER_GET_METHOD_CALIBS_LIST_A AND NOT "DB16000_OPC_UA_TRIGGER_ALARM".CLIENT.U2_STA3_COAXIAL.ALARMS.COMPUTER_GET_METHOD_ANALISIS_LIST_A AND NOT "DB16000_OPC_UA_TRIGGER_ALARM".CLIENT.U2_STA3_COAXIAL.ALARMS.COMPUTER_RELEASE_HANDLE_LIST_A AND NOT "DB16000_OPC_UA_TRIGGER_ALARM".CLIENT.U2_STA3_COAXIAL.ALARMS.COMPUTER_RELEASE_METHOD_CALIBS_LIST_A AND NOT "DB16000_OPC_UA_TRIGGER_ALARM".CLIENT.U2_STA3_COAXIAL.ALARMS.COMPUTER_RELEASE_METHOD_ANALISIS_LIST_A AND NOT "DB16000_OPC_UA_TRIGGER_ALARM".CLIENT.U2_STA3_COAXIAL.ALARMS.COMPUTER_DISCONNECT_A AND NOT "DB16000_OPC_UA_TRIGGER_ALARM".CLIENT.U2_STA3_COAXIAL.ALARMS.CAM_START_LASER_CALIB_CONNECTION_A AND NOT "DB16000_OPC_UA_TRIGGER_ALARM".CLIENT.U2_STA3_COAXIAL.ALARMS.CAM_START_LASER_CALIB_METHOD_WORKING_BLOCKED_A AND NOT "DB16000_OPC_UA_TRIGGER_ALARM".CLIENT.U2_STA3_COAXIAL.ALARMS.CAM_START_NOZZLE_CALIB_CONNECTION_A);
   #ALARM_AUX := NOT ("M_ONE" AND NOT #ALARM_AUX AND NOT "DB16000_OPC_UA_TRIGGER_ALARM".CLIENT.U2_STA3_COAXIAL.ALARMS.CAM_START_NOZZLE_CALIB_METHOD_WORKING_BLOCKED_A AND NOT "DB16000_OPC_UA_TRIGGER_ALARM".CLIENT.U2_STA3_COAXIAL.ALARMS.CAM_START_JET_CALIB_CONNECTION_A AND NOT "DB16000_OPC_UA_TRIGGER_ALARM".CLIENT.U2_STA3_COAXIAL.ALARMS.CAM_START_JET_CALIB_METHOD_WORKING_BLOCKED_A AND NOT "DB16000_OPC_UA_TRIGGER_ALARM".CLIENT.U2_STA3_COAXIAL.ALARMS.CAM_START_CLADD_CALIB_CONNECTION_A AND NOT "DB16000_OPC_UA_TRIGGER_ALARM".CLIENT.U2_STA3_COAXIAL.ALARMS.CAM_START_CLADD_CALIB_METHOD_WORKING_BLOCKED_A AND NOT "DB16000_OPC_UA_TRIGGER_ALARM".CLIENT.U2_STA3_COAXIAL.ALARMS.CAM_START_NOZZLE_ANALISIS_CONNECTION_A AND NOT "DB16000_OPC_UA_TRIGGER_ALARM".CLIENT.U2_STA3_COAXIAL.ALARMS.CAM_START_NOZZLE_ANALISIS_METHOD_WORKING_BLOCKED_A AND NOT "DB16000_OPC_UA_TRIGGER_ALARM".CLIENT.U2_STA3_COAXIAL.ALARMS.CAM_START_JET_ANALISIS_CONNECTION_A AND NOT "DB16000_OPC_UA_TRIGGER_ALARM".CLIENT.U2_STA3_COAXIAL.ALARMS.CAM_START_JET_ANALISIS_METHOD_WORKING_BLOCKED_A AND NOT "DB16000_OPC_UA_TRIGGER_ALARM".CLIENT.U2_STA3_COAXIAL.ALARMS.CAM_START_CLADD_ANALISIS_CONNECTION_A AND NOT "DB16000_OPC_UA_TRIGGER_ALARM".CLIENT.U2_STA3_COAXIAL.ALARMS.CAM_START_CLADD_ANALISIS_METHOD_WORKING_BLOCKED_A);
   #ALARM_AUX := NOT ("M_ONE" AND NOT #ALARM_AUX AND NOT "DB16000_OPC_UA_TRIGGER_ALARM".CLIENT.U2_STA3_COAXIAL.ALARMS.CAM_STOP_METHODS_CONNECTION_A AND NOT "DB16000_OPC_UA_TRIGGER_ALARM".CLIENT.U2_STA3_COAXIAL.ALARMS.CAM_STOP_METHODS_METHOD_WORKING_BLOCKED_A AND NOT "DB16000_OPC_UA_TRIGGER_ALARM".CLIENT.U2_STA3_COAXIAL.ALARMS.RESET_PC_CONNECTION_A AND NOT "DB16000_OPC_UA_TRIGGER_ALARM".CLIENT.U2_STA3_COAXIAL.ALARMS.RESET_PC_METHOD_WORKING_BLOCKED_A AND NOT "DB16000_OPC_UA_TRIGGER_ALARM".CLIENT.U2_STA3_COAXIAL.ALARMS.READ_VARS_CONNECTION_A AND NOT "DB16000_OPC_UA_TRIGGER_ALARM".CLIENT.U2_STA3_COAXIAL.ALARMS.READ_VARS_METHOD_WORKING_BLOCKED_A AND NOT "DB16000_OPC_UA_TRIGGER_ALARM".CLIENT.U2_STA3_COAXIAL.ALARMS.FAILED_CONNECT_CAMERA_A AND NOT "DB16000_OPC_UA_TRIGGER_ALARM".CLIENT.U2_STA3_COAXIAL.ALARMS.FAILED_SET_CAMERA_PARAMETERS_A AND NOT "DB16000_OPC_UA_TRIGGER_ALARM".CLIENT.U2_STA3_COAXIAL.ALARMS.LASER_CALIB_REQUIERED_A AND NOT "DB16000_OPC_UA_TRIGGER_ALARM".CLIENT.U2_STA3_COAXIAL.ALARMS.JET_CALIB_REQUIERED_A AND NOT "DB16000_OPC_UA_TRIGGER_ALARM".CLIENT.U2_STA3_COAXIAL.ALARMS.CLADDING_CALIB_REQUIERED_A);
   #ALARM_AUX := NOT ("M_ONE" AND NOT #ALARM_AUX AND NOT "DB16000_OPC_UA_TRIGGER_ALARM".CLIENT.U2_STA3_COAXIAL.ALARMS.HIGH_NUM_DEAD_PIXELS_A AND NOT "DB16000_OPC_UA_TRIGGER_ALARM".CLIENT.U2_STA3_COAXIAL.ALARMS.CAM_NO_LIGHT_DETECTED_A AND NOT "DB16000_OPC_UA_TRIGGER_ALARM".CLIENT.U2_STA3_COAXIAL.ALARMS.CAM_NO_LASER_DETECTED_A AND NOT "DB16000_OPC_UA_TRIGGER_ALARM".CLIENT.U2_STA3_COAXIAL.ALARMS.CAM_NO_NOZZLE_DETECTED_A AND NOT "DB16000_OPC_UA_TRIGGER_ALARM".CLIENT.U2_STA3_COAXIAL.ALARMS.CAM_NOZZLE_CONTAMINATION_A AND NOT "DB16000_OPC_UA_TRIGGER_ALARM".CLIENT.U2_STA3_COAXIAL.ALARMS.CAM_NO_POWDER_FLOW_DETECTED_A AND NOT "DB16000_OPC_UA_TRIGGER_ALARM".CLIENT.U2_STA3_COAXIAL.ALARMS.CAM_NO_LASER_PATERN_DETECTED_A AND NOT "DB16000_OPC_UA_TRIGGER_ALARM".CLIENT.U2_STA3_COAXIAL.ALARMS.CAM_NOT_ANALYZED_A AND NOT "DB16000_OPC_UA_TRIGGER_ALARM".CLIENT.U2_STA3_COAXIAL.ALARMS.CAM_FAILED_OBTAIN_SCALE_FACTOR_A AND NOT "DB16000_OPC_UA_TRIGGER_ALARM".CLIENT.U2_STA3_COAXIAL.ALARMS.CAM_UNALIGNED_POWDER_FLOW_VORTEX_A AND NOT "DB16000_OPC_UA_TRIGGER_ALARM".CLIENT.U2_STA3_COAXIAL.ALARMS.CAM_JET_MALFUNCTION_A);
   IF NOT ("M_ONE" AND NOT #ALARM_AUX AND NOT "DB16000_OPC_UA_TRIGGER_ALARM".CLIENT.U2_STA3_COAXIAL.ALARMS.CAM_UNCALIBRATED_A AND NOT "DB16000_OPC_UA_TRIGGER_ALARM".CLIENT.U2_STA3_COAXIAL.ALARMS.DMC_STRUCTURE_A AND NOT "DB16000_OPC_UA_TRIGGER_ALARM".CLIENT.U2_STA3_COAXIAL.ALARMS.PLC_PC_MAJOR_VERSIONS_MISMATCH_A AND NOT "DB16000_OPC_UA_TRIGGER_ALARM".CLIENT.U2_STA3_COAXIAL.ALARMS.CAM_NO_MELTPOOL_DETECTED_A AND NOT "DB16000_OPC_UA_TRIGGER_ALARM".CLIENT.U2_STA3_COAXIAL.ALARMS.CAM_NO_DATA_BASE_CONNECTION_A AND NOT "DB16000_OPC_UA_TRIGGER_ALARM".CLIENT.U2_STA3_COAXIAL.ALARMS.CAM_NO_HALO_DETECTED_A AND NOT "DB16000_OPC_UA_TRIGGER_ALARM".CLIENT.U2_STA3_COAXIAL.ALARMS.CAM_STORAGE_ERROR_A AND NOT "DB16000_OPC_UA_TRIGGER_ALARM".CLIENT.U2_STA3_COAXIAL.ALARMS.CAM_INITIALIZING_SENSOR_A AND NOT "DB16000_OPC_UA_TRIGGER_ALARM".CLIENT.U2_STA3_COAXIAL.ALARMS.INVALID_CONFIGURATION_A) THEN
       "DB441_MACHINE_POWDER_ALARM_DECODING".POWDER_ALARMS_GENERAL.ALARM_DECODING := #FC_NUMBER;
       "DB441_MACHINE_POWDER_ALARM_DECODING".POWDER_ALARMS_GENERAL.MP_ALARMS := TRUE;
   END_IF;
END_REGION

REGION Network 108: WARNINGS
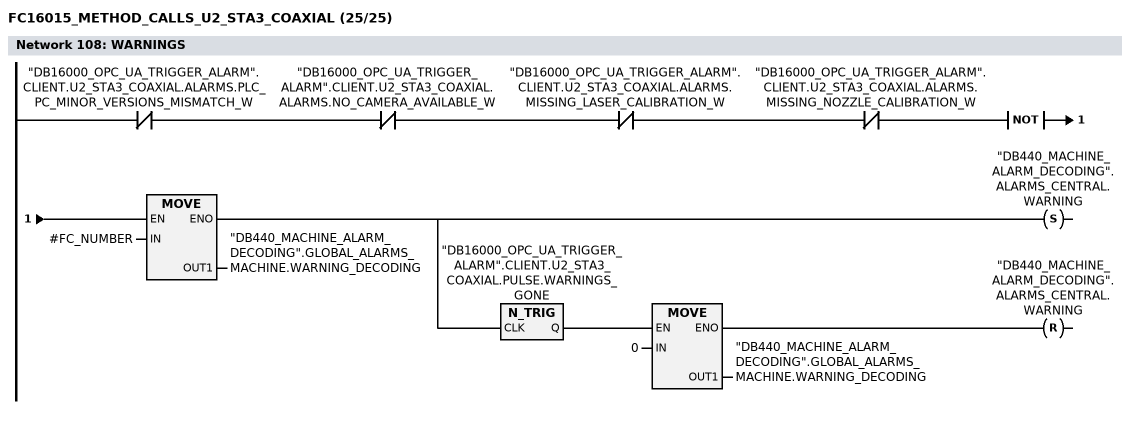
   RUNG wire#powerrail
      I_Contact( "DB16000_OPC_UA_TRIGGER_ALARM".CLIENT.U2_STA3_COAXIAL.ALARMS.PLC_PC_MINOR_VERSIONS_MISMATCH_W )
      I_Contact( "DB16000_OPC_UA_TRIGGER_ALARM".CLIENT.U2_STA3_COAXIAL.ALARMS.NO_CAMERA_AVAILABLE_W )
      I_Contact( "DB16000_OPC_UA_TRIGGER_ALARM".CLIENT.U2_STA3_COAXIAL.ALARMS.MISSING_LASER_CALIBRATION_W )
      I_Contact( "DB16000_OPC_UA_TRIGGER_ALARM".CLIENT.U2_STA3_COAXIAL.ALARMS.MISSING_NOZZLE_CALIBRATION_W )
      Not()
      Move(in := #FC_NUMBER, out1 => "DB440_MACHINE_ALARM_DECODING".GLOBAL_ALARMS_MACHINE.WARNING_DECODING)
      wire#w1
      S_Coil( "DB440_MACHINE_ALARM_DECODING".ALARMS_CENTRAL.WARNING )
   END_RUNG
   RUNG wire#w1
      N_Trig( "DB16000_OPC_UA_TRIGGER_ALARM".CLIENT.U2_STA3_COAXIAL.PULSE.WARNINGS_GONE )
      Move(in := 0, out1 => "DB440_MACHINE_ALARM_DECODING".GLOBAL_ALARMS_MACHINE.WARNING_DECODING)
      R_Coil( "DB440_MACHINE_ALARM_DECODING".ALARMS_CENTRAL.WARNING )
   END_RUNG
   // the same network as SCL:
   #_w1 := NOT (NOT "DB16000_OPC_UA_TRIGGER_ALARM".CLIENT.U2_STA3_COAXIAL.ALARMS.PLC_PC_MINOR_VERSIONS_MISMATCH_W AND NOT "DB16000_OPC_UA_TRIGGER_ALARM".CLIENT.U2_STA3_COAXIAL.ALARMS.NO_CAMERA_AVAILABLE_W AND NOT "DB16000_OPC_UA_TRIGGER_ALARM".CLIENT.U2_STA3_COAXIAL.ALARMS.MISSING_LASER_CALIBRATION_W AND NOT "DB16000_OPC_UA_TRIGGER_ALARM".CLIENT.U2_STA3_COAXIAL.ALARMS.MISSING_NOZZLE_CALIBRATION_W);
   IF #_w1 THEN
       "DB440_MACHINE_ALARM_DECODING".GLOBAL_ALARMS_MACHINE.WARNING_DECODING := #FC_NUMBER;
       "DB440_MACHINE_ALARM_DECODING".ALARMS_CENTRAL.WARNING := TRUE;
   END_IF;
   #_w2 := NOT #_w1 AND "DB16000_OPC_UA_TRIGGER_ALARM".CLIENT.U2_STA3_COAXIAL.PULSE.WARNINGS_GONE;   // falling edge
   "DB16000_OPC_UA_TRIGGER_ALARM".CLIENT.U2_STA3_COAXIAL.PULSE.WARNINGS_GONE := #_w1;
   IF #_w2 THEN
       "DB440_MACHINE_ALARM_DECODING".GLOBAL_ALARMS_MACHINE.WARNING_DECODING := 0;
       "DB440_MACHINE_ALARM_DECODING".ALARMS_CENTRAL.WARNING := FALSE;
   END_IF;
END_REGION
END_FUNCTION
